  [5242] = {x=-104.947, y=80.94, z=66, rx=-180, rz=-143.366, shoulder=lefty, elbow=epositive, wrist=wpositive, fatherId=fReference[0]}
  [5243] = {x=-103.694, y=80.008, z=66, rx=-180, rz=-143.329, shoulder=lefty, elbow=epositive, wrist=wpositive, fatherId=fReference[0]}
  [5244] = {x=-102.442, y=79.076, z=66, rx=-180, rz=-143.293, shoulder=lefty, elbow=epositive, wrist=wpositive, fatherId=fReference[0]}
  [5245] = {x=-101.19, y=78.143, z=66, rx=-180, rz=-143.258, shoulder=lefty, elbow=epositive, wrist=wpositive, fatherId=fReference[0]}
  [5246] = {x=-99.938, y=77.208, z=66, rx=-180, rz=-143.223, shoulder=lefty, elbow=epositive, wrist=wpositive, fatherId=fReference[0]}
  [5247] = {x=-98.687, y=76.273, z=66, rx=-180, rz=-143.188, shoulder=lefty, elbow=epositive, wrist=wpositive, fatherId=fReference[0]}
  [5248] = {x=-97.437, y=75.337, z=66, rx=180, rz=-143.154, shoulder=lefty, elbow=epositive, wrist=wpositive, fatherId=fReference[0]}
  [5249] = {x=-96.186, y=74.4, z=66, rx=180, rz=-143.12, shoulder=lefty, elbow=epositive, wrist=wpositive, fatherId=fReference[0]}
  [5250] = {x=-94.936, y=73.462, z=66, rx=180, rz=-143.087, shoulder=lefty, elbow=epositive, wrist=wpositive, fatherId=fReference[0]}
  [5251] = {x=-93.686, y=72.523, z=66, rx=-180, rz=-143.054, shoulder=lefty, elbow=epositive, wrist=wpositive, fatherId=fReference[0]}
  [5252] = {x=-92.437, y=71.584, z=66, rx=180, rz=-143.022, shoulder=lefty, elbow=epositive, wrist=wpositive, fatherId=fReference[0]}
  [5253] = {x=-91.188, y=70.643, z=66, rx=-180, rz=-142.99, shoulder=lefty, elbow=epositive, wrist=wpositive, fatherId=fReference[0]}
  [5254] = {x=-89.939, y=69.702, z=66, rx=-180, rz=-142.959, shoulder=lefty, elbow=epositive, wrist=wpositive, fatherId=fReference[0]}
  [5255] = {x=-88.691, y=68.76, z=66, rx=-180, rz=-142.928, shoulder=lefty, elbow=epositive, wrist=wpositive, fatherId=fReference[0]}
  [5256] = {x=-87.443, y=67.817, z=66, rx=-180, rz=-142.897, shoulder=lefty, elbow=epositive, wrist=wpositive, fatherId=fReference[0]}
  [5257] = {x=-86.195, y=66.873, z=66, rx=180, rz=-142.867, shoulder=lefty, elbow=epositive, wrist=wpositive, fatherId=fReference[0]}
  [5258] = {x=-84.948, y=65.929, z=66, rx=-180, rz=-142.838, shoulder=lefty, elbow=epositive, wrist=wpositive, fatherId=fReference[0]}
  [5259] = {x=-83.701, y=64.984, z=66, rx=180, rz=-142.809, shoulder=lefty, elbow=epositive, wrist=wpositive, fatherId=fReference[0]}
  [5260] = {x=-82.454, y=64.038, z=66, rx=180, rz=-142.78, shoulder=lefty, elbow=epositive, wrist=wpositive, fatherId=fReference[0]}
  [5261] = {x=-81.208, y=63.091, z=66, rx=-180, rz=-142.752, shoulder=lefty, elbow=epositive, wrist=wpositive, fatherId=fReference[0]}
  [5262] = {x=-79.962, y=62.143, z=66, rx=-180, rz=-142.724, shoulder=lefty, elbow=epositive, wrist=wpositive, fatherId=fReference[0]}
  [5263] = {x=-78.716, y=61.195, z=66, rx=-180, rz=-142.697, shoulder=lefty, elbow=epositive, wrist=wpositive, fatherId=fReference[0]}
  [5264] = {x=-77.47, y=60.246, z=66, rx=-180, rz=-142.67, shoulder=lefty, elbow=epositive, wrist=wpositive, fatherId=fReference[0]}
  [5265] = {x=-76.225, y=59.297, z=66, rx=180, rz=-142.644, shoulder=lefty, elbow=epositive, wrist=wpositive, fatherId=fReference[0]}
  [5266] = {x=-74.98, y=58.346, z=66, rx=-180, rz=-142.618, shoulder=lefty, elbow=epositive, wrist=wpositive, fatherId=fReference[0]}
  [5267] = {x=-73.736, y=57.395, z=66, rx=180, rz=-142.592, shoulder=lefty, elbow=epositive, wrist=wpositive, fatherId=fReference[0]}
  [5268] = {x=-72.491, y=56.444, z=66, rx=-180, rz=-142.567, shoulder=lefty, elbow=epositive, wrist=wpositive, fatherId=fReference[0]}
  [5269] = {x=-71.247, y=55.491, z=66, rx=180, rz=-142.543, shoulder=lefty, elbow=epositive, wrist=wpositive, fatherId=fReference[0]}
  [5270] = {x=-70.003, y=54.538, z=66, rx=180, rz=-142.518, shoulder=lefty, elbow=epositive, wrist=wpositive, fatherId=fReference[0]}
  [5271] = {x=-68.76, y=53.585, z=66, rx=-180, rz=-142.495, shoulder=lefty, elbow=epositive, wrist=wpositive, fatherId=fReference[0]}
  [5272] = {x=-67.516, y=52.63, z=66, rx=-180, rz=-142.471, shoulder=lefty, elbow=epositive, wrist=wpositive, fatherId=fReference[0]}
  [5273] = {x=-66.273, y=51.676, z=66, rx=-180, rz=-142.449, shoulder=lefty, elbow=epositive, wrist=wpositive, fatherId=fReference[0]}
  [5274] = {x=-65.03, y=50.72, z=66, rx=-180, rz=-142.426, shoulder=lefty, elbow=epositive, wrist=wpositive, fatherId=fReference[0]}
  [5275] = {x=-63.788, y=49.764, z=66, rx=-180, rz=-142.404, shoulder=lefty, elbow=epositive, wrist=wpositive, fatherId=fReference[0]}
  [5276] = {x=-62.545, y=48.808, z=66, rx=-180, rz=-142.383, shoulder=lefty, elbow=epositive, wrist=wpositive, fatherId=fReference[0]}
  [5277] = {x=-61.303, y=47.85, z=66, rx=-180, rz=-142.362, shoulder=lefty, elbow=epositive, wrist=wpositive, fatherId=fReference[0]}
  [5278] = {x=-60.061, y=46.893, z=66, rx=-180, rz=-142.341, shoulder=lefty, elbow=epositive, wrist=wpositive, fatherId=fReference[0]}
  [5279] = {x=-58.82, y=45.934, z=66, rx=180, rz=-142.321, shoulder=lefty, elbow=epositive, wrist=wpositive, fatherId=fReference[0]}
  [5280] = {x=-57.578, y=44.976, z=66, rx=-180, rz=-142.301, shoulder=lefty, elbow=epositive, wrist=wpositive, fatherId=fReference[0]}
  [5281] = {x=-56.337, y=44.016, z=66, rx=180, rz=-142.282, shoulder=lefty, elbow=epositive, wrist=wpositive, fatherId=fReference[0]}
  [5282] = {x=-55.096, y=43.057, z=66, rx=-180, rz=-142.263, shoulder=lefty, elbow=epositive, wrist=wpositive, fatherId=fReference[0]}
  [5283] = {x=-53.855, y=42.096, z=66, rx=-180, rz=-142.244, shoulder=lefty, elbow=epositive, wrist=wpositive, fatherId=fReference[0]}
  [5284] = {x=-52.615, y=41.135, z=66, rx=-180, rz=-142.226, shoulder=lefty, elbow=epositive, wrist=wpositive, fatherId=fReference[0]}
  [5285] = {x=-51.374, y=40.174, z=66, rx=-180, rz=-142.209, shoulder=lefty, elbow=epositive, wrist=wpositive, fatherId=fReference[0]}
  [5286] = {x=-50.134, y=39.212, z=66, rx=-180, rz=-142.192, shoulder=lefty, elbow=epositive, wrist=wpositive, fatherId=fReference[0]}
  [5287] = {x=-48.894, y=38.25, z=66, rx=-180, rz=-142.175, shoulder=lefty, elbow=epositive, wrist=wpositive, fatherId=fReference[0]}
  [5288] = {x=-47.654, y=37.288, z=66, rx=-180, rz=-142.159, shoulder=lefty, elbow=epositive, wrist=wpositive, fatherId=fReference[0]}
  [5289] = {x=-46.414, y=36.325, z=66, rx=180, rz=-142.143, shoulder=lefty, elbow=epositive, wrist=wpositive, fatherId=fReference[0]}
  [5290] = {x=-45.175, y=35.361, z=66, rx=-180, rz=-142.127, shoulder=lefty, elbow=epositive, wrist=wpositive, fatherId=fReference[0]}
  [5291] = {x=-43.935, y=34.397, z=66, rx=180, rz=-142.112, shoulder=lefty, elbow=epositive, wrist=wpositive, fatherId=fReference[0]}
  [5292] = {x=-42.696, y=33.433, z=66, rx=180, rz=-142.098, shoulder=lefty, elbow=epositive, wrist=wpositive, fatherId=fReference[0]}
  [5293] = {x=-41.457, y=32.468, z=66, rx=180, rz=-142.083, shoulder=lefty, elbow=epositive, wrist=wpositive, fatherId=fReference[0]}
  [5294] = {x=-40.218, y=31.503, z=66, rx=-180, rz=-142.07, shoulder=lefty, elbow=epositive, wrist=wpositive, fatherId=fReference[0]}
  [5295] = {x=-38.979, y=30.538, z=66, rx=180, rz=-142.056, shoulder=lefty, elbow=epositive, wrist=wpositive, fatherId=fReference[0]}
  [5296] = {x=-37.74, y=29.572, z=66, rx=-180, rz=-142.044, shoulder=lefty, elbow=epositive, wrist=wpositive, fatherId=fReference[0]}
  [5297] = {x=-36.502, y=28.606, z=66, rx=-180, rz=-142.031, shoulder=lefty, elbow=epositive, wrist=wpositive, fatherId=fReference[0]}
  [5298] = {x=-35.263, y=27.639, z=66, rx=180, rz=-142.019, shoulder=lefty, elbow=epositive, wrist=wpositive, fatherId=fReference[0]}
  [5299] = {x=-34.025, y=26.672, z=66, rx=-180, rz=-142.007, shoulder=lefty, elbow=epositive, wrist=wpositive, fatherId=fReference[0]}
  [5300] = {x=-32.787, y=25.705, z=66, rx=-180, rz=-141.996, shoulder=lefty, elbow=epositive, wrist=wpositive, fatherId=fReference[0]}
  [5301] = {x=-31.549, y=24.738, z=66, rx=180, rz=-141.985, shoulder=lefty, elbow=epositive, wrist=wpositive, fatherId=fReference[0]}
  [5302] = {x=-30.311, y=23.77, z=66, rx=180, rz=-141.975, shoulder=lefty, elbow=epositive, wrist=wpositive, fatherId=fReference[0]}
  [5303] = {x=-29.073, y=22.802, z=66, rx=180, rz=-141.965, shoulder=lefty, elbow=epositive, wrist=wpositive, fatherId=fReference[0]}
  [5304] = {x=-27.835, y=21.834, z=66, rx=-180, rz=-141.956, shoulder=lefty, elbow=epositive, wrist=wpositive, fatherId=fReference[0]}
  [5305] = {x=-26.597, y=20.865, z=66, rx=-180, rz=-141.947, shoulder=lefty, elbow=epositive, wrist=wpositive, fatherId=fReference[0]}
  [5306] = {x=-25.36, y=19.896, z=66, rx=180, rz=-141.938, shoulder=lefty, elbow=epositive, wrist=wpositive, fatherId=fReference[0]}
  [5307] = {x=-24.122, y=18.927, z=66, rx=-180, rz=-141.93, shoulder=lefty, elbow=epositive, wrist=wpositive, fatherId=fReference[0]}
  [5308] = {x=-22.885, y=17.958, z=66, rx=180, rz=-141.922, shoulder=lefty, elbow=epositive, wrist=wpositive, fatherId=fReference[0]}
  [5309] = {x=-21.647, y=16.988, z=66, rx=-180, rz=-141.915, shoulder=lefty, elbow=epositive, wrist=wpositive, fatherId=fReference[0]}
  [5310] = {x=-20.41, y=16.019, z=66, rx=-180, rz=-141.908, shoulder=lefty, elbow=epositive, wrist=wpositive, fatherId=fReference[0]}
  [5311] = {x=-19.172, y=15.049, z=66, rx=-180, rz=-141.901, shoulder=lefty, elbow=epositive, wrist=wpositive, fatherId=fReference[0]}
  [5312] = {x=-17.935, y=14.079, z=66, rx=-180, rz=-141.895, shoulder=lefty, elbow=epositive, wrist=wpositive, fatherId=fReference[0]}
  [5313] = {x=-16.698, y=13.109, z=66, rx=180, rz=-141.889, shoulder=lefty, elbow=epositive, wrist=wpositive, fatherId=fReference[0]}
  [5314] = {x=-15.461, y=12.138, z=66, rx=-180, rz=-141.884, shoulder=lefty, elbow=epositive, wrist=wpositive, fatherId=fReference[0]}
  [5315] = {x=-14.224, y=11.168, z=66, rx=-180, rz=-141.879, shoulder=lefty, elbow=epositive, wrist=wpositive, fatherId=fReference[0]}
  [5316] = {x=-12.987, y=10.197, z=66, rx=-180, rz=-141.875, shoulder=lefty, elbow=epositive, wrist=wpositive, fatherId=fReference[0]}
  [5317] = {x=-11.75, y=9.226, z=66, rx=-180, rz=-141.871, shoulder=lefty, elbow=epositive, wrist=wpositive, fatherId=fReference[0]}
  [5318] = {x=-10.513, y=8.255, z=66, rx=-180, rz=-141.867, shoulder=lefty, elbow=epositive, wrist=wpositive, fatherId=fReference[0]}
  [5319] = {x=-9.276, y=7.284, z=66, rx=-180, rz=-141.864, shoulder=lefty, elbow=epositive, wrist=wpositive, fatherId=fReference[0]}
  [5320] = {x=-8.039, y=6.313, z=66, rx=180, rz=-141.862, shoulder=lefty, elbow=epositive, wrist=wpositive, fatherId=fReference[0]}
  [5321] = {x=-6.802, y=5.342, z=66, rx=-180, rz=-141.859, shoulder=lefty, elbow=epositive, wrist=wpositive, fatherId=fReference[0]}
  [5322] = {x=-5.565, y=4.37, z=66, rx=180, rz=-141.857, shoulder=lefty, elbow=epositive, wrist=wpositive, fatherId=fReference[0]}
  [5323] = {x=-4.328, y=3.399, z=66, rx=-180, rz=-141.856, shoulder=lefty, elbow=epositive, wrist=wpositive, fatherId=fReference[0]}
  [5324] = {x=-3.091, y=2.427, z=66, rx=-180, rz=-141.855, shoulder=lefty, elbow=epositive, wrist=wpositive, fatherId=fReference[0]}
  [5325] = {x=-1.854, y=1.456, z=66, rx=180, rz=-141.854, shoulder=lefty, elbow=epositive, wrist=wpositive, fatherId=fReference[0]}
  [5326] = {x=-0.617, y=0.484, z=66, rx=180, rz=-141.854, shoulder=lefty, elbow=epositive, wrist=wpositive, fatherId=fReference[0]}
  [5327] = {x=0.62, y=-0.487, z=66, rx=180, rz=-141.854, shoulder=lefty, elbow=epositive, wrist=wpositive, fatherId=fReference[0]}
  [5328] = {x=1.857, y=-1.459, z=66, rx=-180, rz=-141.855, shoulder=lefty, elbow=epositive, wrist=wpositive, fatherId=fReference[0]}
  [5329] = {x=3.094, y=-2.43, z=66, rx=180, rz=-141.856, shoulder=lefty, elbow=epositive, wrist=wpositive, fatherId=fReference[0]}
  [5330] = {x=4.331, y=-3.402, z=66, rx=-180, rz=-141.857, shoulder=lefty, elbow=epositive, wrist=wpositive, fatherId=fReference[0]}
  [5331] = {x=5.568, y=-4.373, z=66, rx=-180, rz=-141.859, shoulder=lefty, elbow=epositive, wrist=wpositive, fatherId=fReference[0]}
  [5332] = {x=6.805, y=-5.345, z=66, rx=180, rz=-141.862, shoulder=lefty, elbow=epositive, wrist=wpositive, fatherId=fReference[0]}
  [5333] = {x=8.043, y=-6.316, z=66, rx=180, rz=-141.864, shoulder=lefty, elbow=epositive, wrist=wpositive, fatherId=fReference[0]}
  [5334] = {x=9.28, y=-7.287, z=66, rx=180, rz=-141.867, shoulder=lefty, elbow=epositive, wrist=wpositive, fatherId=fReference[0]}
  [5335] = {x=10.517, y=-8.259, z=66, rx=180, rz=-141.871, shoulder=lefty, elbow=epositive, wrist=wpositive, fatherId=fReference[0]}
  [5336] = {x=11.754, y=-9.23, z=66, rx=-180, rz=-141.875, shoulder=lefty, elbow=epositive, wrist=wpositive, fatherId=fReference[0]}
  [5337] = {x=12.992, y=-10.201, z=66, rx=-180, rz=-141.879, shoulder=lefty, elbow=epositive, wrist=wpositive, fatherId=fReference[0]}
  [5338] = {x=14.229, y=-11.172, z=66, rx=180, rz=-141.884, shoulder=lefty, elbow=epositive, wrist=wpositive, fatherId=fReference[0]}
  [5339] = {x=15.467, y=-12.143, z=66, rx=-180, rz=-141.89, shoulder=lefty, elbow=epositive, wrist=wpositive, fatherId=fReference[0]}
  [5340] = {x=16.704, y=-13.113, z=66, rx=180, rz=-141.895, shoulder=lefty, elbow=epositive, wrist=wpositive, fatherId=fReference[0]}
  [5341] = {x=17.942, y=-14.084, z=66, rx=180, rz=-141.901, shoulder=lefty, elbow=epositive, wrist=wpositive, fatherId=fReference[0]}
  [5342] = {x=19.179, y=-15.054, z=66, rx=-180, rz=-141.908, shoulder=lefty, elbow=epositive, wrist=wpositive, fatherId=fReference[0]}
  [5343] = {x=20.417, y=-16.025, z=66, rx=-180, rz=-141.915, shoulder=lefty, elbow=epositive, wrist=wpositive, fatherId=fReference[0]}
  [5344] = {x=21.655, y=-16.995, z=66, rx=180, rz=-141.922, shoulder=lefty, elbow=epositive, wrist=wpositive, fatherId=fReference[0]}
  [5345] = {x=22.893, y=-17.965, z=66, rx=180, rz=-141.93, shoulder=lefty, elbow=epositive, wrist=wpositive, fatherId=fReference[0]}
  [5346] = {x=24.131, y=-18.934, z=66, rx=-180, rz=-141.938, shoulder=lefty, elbow=epositive, wrist=wpositive, fatherId=fReference[0]}
  [5347] = {x=25.369, y=-19.904, z=66, rx=-180, rz=-141.947, shoulder=lefty, elbow=epositive, wrist=wpositive, fatherId=fReference[0]}
  [5348] = {x=26.607, y=-20.873, z=66, rx=180, rz=-141.956, shoulder=lefty, elbow=epositive, wrist=wpositive, fatherId=fReference[0]}
  [5349] = {x=27.846, y=-21.842, z=66, rx=-180, rz=-141.965, shoulder=lefty, elbow=epositive, wrist=wpositive, fatherId=fReference[0]}
  [5350] = {x=29.084, y=-22.811, z=66, rx=-180, rz=-141.975, shoulder=lefty, elbow=epositive, wrist=wpositive, fatherId=fReference[0]}
  [5351] = {x=30.323, y=-23.779, z=66, rx=-180, rz=-141.986, shoulder=lefty, elbow=epositive, wrist=wpositive, fatherId=fReference[0]}
  [5352] = {x=31.561, y=-24.748, z=66, rx=-180, rz=-141.996, shoulder=lefty, elbow=epositive, wrist=wpositive, fatherId=fReference[0]}
  [5353] = {x=32.8, y=-25.716, z=66, rx=-180, rz=-142.008, shoulder=lefty, elbow=epositive, wrist=wpositive, fatherId=fReference[0]}
  [5354] = {x=34.039, y=-26.683, z=66, rx=180, rz=-142.019, shoulder=lefty, elbow=epositive, wrist=wpositive, fatherId=fReference[0]}
  [5355] = {x=35.278, y=-27.651, z=66, rx=-180, rz=-142.031, shoulder=lefty, elbow=epositive, wrist=wpositive, fatherId=fReference[0]}
  [5356] = {x=36.517, y=-28.618, z=66, rx=180, rz=-142.044, shoulder=lefty, elbow=epositive, wrist=wpositive, fatherId=fReference[0]}
  [5357] = {x=37.757, y=-29.585, z=66, rx=-180, rz=-142.057, shoulder=lefty, elbow=epositive, wrist=wpositive, fatherId=fReference[0]}
  [5358] = {x=38.996, y=-30.551, z=66, rx=-180, rz=-142.07, shoulder=lefty, elbow=epositive, wrist=wpositive, fatherId=fReference[0]}
  [5359] = {x=40.236, y=-31.517, z=66, rx=-180, rz=-142.084, shoulder=lefty, elbow=epositive, wrist=wpositive, fatherId=fReference[0]}
  [5360] = {x=41.476, y=-32.483, z=66, rx=-180, rz=-142.098, shoulder=lefty, elbow=epositive, wrist=wpositive, fatherId=fReference[0]}
  [5361] = {x=42.715, y=-33.448, z=66, rx=180, rz=-142.113, shoulder=lefty, elbow=epositive, wrist=wpositive, fatherId=fReference[0]}
  [5362] = {x=43.956, y=-34.413, z=66, rx=180, rz=-142.128, shoulder=lefty, elbow=epositive, wrist=wpositive, fatherId=fReference[0]}
  [5363] = {x=45.196, y=-35.377, z=66, rx=-180, rz=-142.143, shoulder=lefty, elbow=epositive, wrist=wpositive, fatherId=fReference[0]}
  [5364] = {x=46.436, y=-36.342, z=66, rx=-180, rz=-142.159, shoulder=lefty, elbow=epositive, wrist=wpositive, fatherId=fReference[0]}
  [5365] = {x=47.677, y=-37.305, z=66, rx=-180, rz=-142.175, shoulder=lefty, elbow=epositive, wrist=wpositive, fatherId=fReference[0]}
  [5366] = {x=48.917, y=-38.269, z=66, rx=180, rz=-142.192, shoulder=lefty, elbow=epositive, wrist=wpositive, fatherId=fReference[0]}
  [5367] = {x=50.158, y=-39.231, z=66, rx=180, rz=-142.209, shoulder=lefty, elbow=epositive, wrist=wpositive, fatherId=fReference[0]}
  [5368] = {x=51.399, y=-40.194, z=66, rx=180, rz=-142.227, shoulder=lefty, elbow=epositive, wrist=wpositive, fatherId=fReference[0]}
  [5369] = {x=52.641, y=-41.156, z=66, rx=-180, rz=-142.245, shoulder=lefty, elbow=epositive, wrist=wpositive, fatherId=fReference[0]}
  [5370] = {x=53.882, y=-42.117, z=66, rx=180, rz=-142.263, shoulder=lefty, elbow=epositive, wrist=wpositive, fatherId=fReference[0]}
  [5371] = {x=55.124, y=-43.078, z=66, rx=180, rz=-142.282, shoulder=lefty, elbow=epositive, wrist=wpositive, fatherId=fReference[0]}
  [5372] = {x=56.366, y=-44.038, z=66, rx=-180, rz=-142.302, shoulder=lefty, elbow=epositive, wrist=wpositive, fatherId=fReference[0]}
  [5373] = {x=57.608, y=-44.998, z=66, rx=180, rz=-142.321, shoulder=lefty, elbow=epositive, wrist=wpositive, fatherId=fReference[0]}
  [5374] = {x=58.85, y=-45.958, z=66, rx=-180, rz=-142.342, shoulder=lefty, elbow=epositive, wrist=wpositive, fatherId=fReference[0]}
  [5375] = {x=60.092, y=-46.916, z=66, rx=-180, rz=-142.362, shoulder=lefty, elbow=epositive, wrist=wpositive, fatherId=fReference[0]}
  [5376] = {x=61.335, y=-47.875, z=66, rx=180, rz=-142.383, shoulder=lefty, elbow=epositive, wrist=wpositive, fatherId=fReference[0]}
  [5377] = {x=62.578, y=-48.832, z=66, rx=-180, rz=-142.405, shoulder=lefty, elbow=epositive, wrist=wpositive, fatherId=fReference[0]}
  [5378] = {x=63.821, y=-49.79, z=66, rx=-180, rz=-142.427, shoulder=lefty, elbow=epositive, wrist=wpositive, fatherId=fReference[0]}
  [5379] = {x=65.064, y=-50.746, z=66, rx=180, rz=-142.449, shoulder=lefty, elbow=epositive, wrist=wpositive, fatherId=fReference[0]}
  [5380] = {x=66.308, y=-51.702, z=66, rx=-180, rz=-142.472, shoulder=lefty, elbow=epositive, wrist=wpositive, fatherId=fReference[0]}
  [5381] = {x=67.551, y=-52.657, z=66, rx=-180, rz=-142.496, shoulder=lefty, elbow=epositive, wrist=wpositive, fatherId=fReference[0]}
  [5382] = {x=68.795, y=-53.612, z=66, rx=-180, rz=-142.519, shoulder=lefty, elbow=epositive, wrist=wpositive, fatherId=fReference[0]}
  [5383] = {x=70.04, y=-54.566, z=66, rx=180, rz=-142.543, shoulder=lefty, elbow=epositive, wrist=wpositive, fatherId=fReference[0]}
  [5384] = {x=71.284, y=-55.519, z=66, rx=-180, rz=-142.568, shoulder=lefty, elbow=epositive, wrist=wpositive, fatherId=fReference[0]}
  [5385] = {x=72.529, y=-56.472, z=66, rx=-180, rz=-142.593, shoulder=lefty, elbow=epositive, wrist=wpositive, fatherId=fReference[0]}
  [5386] = {x=73.774, y=-57.424, z=66, rx=180, rz=-142.619, shoulder=lefty, elbow=epositive, wrist=wpositive, fatherId=fReference[0]}
  [5387] = {x=75.019, y=-58.376, z=66, rx=-180, rz=-142.645, shoulder=lefty, elbow=epositive, wrist=wpositive, fatherId=fReference[0]}
  [5388] = {x=76.264, y=-59.326, z=66, rx=-180, rz=-142.671, shoulder=lefty, elbow=epositive, wrist=wpositive, fatherId=fReference[0]}
  [5389] = {x=77.51, y=-60.276, z=66, rx=-180, rz=-142.698, shoulder=lefty, elbow=epositive, wrist=wpositive, fatherId=fReference[0]}
  [5390] = {x=78.756, y=-61.226, z=66, rx=-180, rz=-142.725, shoulder=lefty, elbow=epositive, wrist=wpositive, fatherId=fReference[0]}
  [5391] = {x=80.002, y=-62.174, z=66, rx=180, rz=-142.753, shoulder=lefty, elbow=epositive, wrist=wpositive, fatherId=fReference[0]}
  [5392] = {x=81.249, y=-63.122, z=66, rx=-180, rz=-142.781, shoulder=lefty, elbow=epositive, wrist=wpositive, fatherId=fReference[0]}
  [5393] = {x=82.496, y=-64.069, z=66, rx=180, rz=-142.81, shoulder=lefty, elbow=epositive, wrist=wpositive, fatherId=fReference[0]}
  [5394] = {x=83.743, y=-65.015, z=66, rx=180, rz=-142.839, shoulder=lefty, elbow=epositive, wrist=wpositive, fatherId=fReference[0]}
  [5395] = {x=84.99, y=-65.961, z=66, rx=-180, rz=-142.868, shoulder=lefty, elbow=epositive, wrist=wpositive, fatherId=fReference[0]}
  [5396] = {x=86.238, y=-66.905, z=66, rx=-180, rz=-142.898, shoulder=lefty, elbow=epositive, wrist=wpositive, fatherId=fReference[0]}
  [5397] = {x=87.486, y=-67.849, z=66, rx=-180, rz=-142.929, shoulder=lefty, elbow=epositive, wrist=wpositive, fatherId=fReference[0]}
  [5398] = {x=88.734, y=-68.792, z=66, rx=-180, rz=-142.96, shoulder=lefty, elbow=epositive, wrist=wpositive, fatherId=fReference[0]}
  [5399] = {x=89.982, y=-69.734, z=66, rx=-180, rz=-142.991, shoulder=lefty, elbow=epositive, wrist=wpositive, fatherId=fReference[0]}
  [5400] = {x=91.231, y=-70.676, z=66, rx=-180, rz=-143.023, shoulder=lefty, elbow=epositive, wrist=wpositive, fatherId=fReference[0]}
  [5401] = {x=92.48, y=-71.616, z=66, rx=180, rz=-143.055, shoulder=lefty, elbow=epositive, wrist=wpositive, fatherId=fReference[0]}
  [5402] = {x=93.73, y=-72.556, z=66, rx=-180, rz=-143.088, shoulder=lefty, elbow=epositive, wrist=wpositive, fatherId=fReference[0]}
  [5403] = {x=94.979, y=-73.495, z=66, rx=-180, rz=-143.121, shoulder=lefty, elbow=epositive, wrist=wpositive, fatherId=fReference[0]}
  [5404] = {x=96.23, y=-74.432, z=66, rx=-180, rz=-143.155, shoulder=lefty, elbow=epositive, wrist=wpositive, fatherId=fReference[0]}
  [5405] = {x=97.48, y=-75.369, z=66, rx=180, rz=-143.189, shoulder=lefty, elbow=epositive, wrist=wpositive, fatherId=fReference[0]}
  [5406] = {x=98.731, y=-76.305, z=66, rx=180, rz=-143.224, shoulder=lefty, elbow=epositive, wrist=wpositive, fatherId=fReference[0]}
  [5407] = {x=99.982, y=-77.24, z=66, rx=-180, rz=-143.259, shoulder=lefty, elbow=epositive, wrist=wpositive, fatherId=fReference[0]}
  [5408] = {x=101.233, y=-78.175, z=66, rx=180, rz=-143.294, shoulder=lefty, elbow=epositive, wrist=wpositive, fatherId=fReference[0]}
  [5409] = {x=102.485, y=-79.108, z=66, rx=-180, rz=-143.33, shoulder=lefty, elbow=epositive, wrist=wpositive, fatherId=fReference[0]}
  [5410] = {x=103.737, y=-80.04, z=66, rx=-180, rz=-143.367, shoulder=lefty, elbow=epositive, wrist=wpositive, fatherId=fReference[0]}
  [5411] = {x=104.989, y=-80.971, z=66, rx=180, rz=-143.404, shoulder=lefty, elbow=epositive, wrist=wpositive, fatherId=fReference[0]}
  [5412] = {x=106.242, y=-81.901, z=66, rx=180, rz=-143.441, shoulder=lefty, elbow=epositive, wrist=wpositive, fatherId=fReference[0]}
  [5413] = {x=107.495, y=-82.831, z=66, rx=180, rz=-143.479, shoulder=lefty, elbow=epositive, wrist=wpositive, fatherId=fReference[0]}
  [5414] = {x=108.748, y=-83.759, z=66, rx=-180, rz=-143.517, shoulder=lefty, elbow=epositive, wrist=wpositive, fatherId=fReference[0]}
  [5415] = {x=110.002, y=-84.686, z=66, rx=-180, rz=-143.556, shoulder=lefty, elbow=epositive, wrist=wpositive, fatherId=fReference[0]}
  [5416] = {x=111.256, y=-85.612, z=66, rx=-180, rz=-143.596, shoulder=lefty, elbow=epositive, wrist=wpositive, fatherId=fReference[0]}
  [5417] = {x=112.511, y=-86.537, z=66, rx=180, rz=-143.635, shoulder=lefty, elbow=epositive, wrist=wpositive, fatherId=fReference[0]}
  [5418] = {x=113.766, y=-87.461, z=66, rx=-180, rz=-143.676, shoulder=lefty, elbow=epositive, wrist=wpositive, fatherId=fReference[0]}
  [5419] = {x=115.021, y=-88.384, z=66, rx=-180, rz=-143.716, shoulder=lefty, elbow=epositive, wrist=wpositive, fatherId=fReference[0]}
  [5420] = {x=116.277, y=-89.306, z=66, rx=-180, rz=-143.758, shoulder=lefty, elbow=epositive, wrist=wpositive, fatherId=fReference[0]}
  [5421] = {x=117.533, y=-90.227, z=66, rx=180, rz=-143.799, shoulder=lefty, elbow=epositive, wrist=wpositive, fatherId=fReference[0]}
  [5422] = {x=118.789, y=-91.146, z=66, rx=180, rz=-143.842, shoulder=lefty, elbow=epositive, wrist=wpositive, fatherId=fReference[0]}
  [5423] = {x=120.046, y=-92.065, z=66, rx=180, rz=-143.884, shoulder=lefty, elbow=epositive, wrist=wpositive, fatherId=fReference[0]}
  [5424] = {x=121.304, y=-92.982, z=66, rx=180, rz=-143.927, shoulder=lefty, elbow=epositive, wrist=wpositive, fatherId=fReference[0]}
  [5425] = {x=122.561, y=-93.898, z=66, rx=180, rz=-143.971, shoulder=lefty, elbow=epositive, wrist=wpositive, fatherId=fReference[0]}
  [5426] = {x=123.819, y=-94.813, z=66, rx=-180, rz=-144.015, shoulder=lefty, elbow=epositive, wrist=wpositive, fatherId=fReference[0]}
  [5427] = {x=125.078, y=-95.727, z=66, rx=-180, rz=-144.06, shoulder=lefty, elbow=epositive, wrist=wpositive, fatherId=fReference[0]}
  [5428] = {x=126.337, y=-96.64, z=66, rx=180, rz=-144.105, shoulder=lefty, elbow=epositive, wrist=wpositive, fatherId=fReference[0]}
  [5429] = {x=127.596, y=-97.551, z=66, rx=-180, rz=-144.151, shoulder=lefty, elbow=epositive, wrist=wpositive, fatherId=fReference[0]}
  [5430] = {x=128.856, y=-98.461, z=66, rx=180, rz=-144.197, shoulder=lefty, elbow=epositive, wrist=wpositive, fatherId=fReference[0]}
  [5431] = {x=130.116, y=-99.37, z=66, rx=180, rz=-144.243, shoulder=lefty, elbow=epositive, wrist=wpositive, fatherId=fReference[0]}
  [5432] = {x=131.376, y=-100.278, z=66, rx=-180, rz=-144.291, shoulder=lefty, elbow=epositive, wrist=wpositive, fatherId=fReference[0]}
  [5433] = {x=132.637, y=-101.185, z=66, rx=-180, rz=-144.338, shoulder=lefty, elbow=epositive, wrist=wpositive, fatherId=fReference[0]}
  [5434] = {x=133.899, y=-102.09, z=66, rx=-180, rz=-144.386, shoulder=lefty, elbow=epositive, wrist=wpositive, fatherId=fReference[0]}
  [5435] = {x=135.161, y=-102.994, z=66, rx=-180, rz=-144.435, shoulder=lefty, elbow=epositive, wrist=wpositive, fatherId=fReference[0]}
  [5436] = {x=136.423, y=-103.896, z=66, rx=180, rz=-144.484, shoulder=lefty, elbow=epositive, wrist=wpositive, fatherId=fReference[0]}
  [5437] = {x=137.686, y=-104.798, z=66, rx=-180, rz=-144.534, shoulder=lefty, elbow=epositive, wrist=wpositive, fatherId=fReference[0]}
  [5438] = {x=138.949, y=-105.698, z=66, rx=180, rz=-144.584, shoulder=lefty, elbow=epositive, wrist=wpositive, fatherId=fReference[0]}
  [5439] = {x=140.213, y=-106.596, z=66, rx=180, rz=-144.634, shoulder=lefty, elbow=epositive, wrist=wpositive, fatherId=fReference[0]}
  [5440] = {x=141.477, y=-107.494, z=66, rx=180, rz=-144.686, shoulder=lefty, elbow=epositive, wrist=wpositive, fatherId=fReference[0]}
  [5441] = {x=142.742, y=-108.389, z=66, rx=-180, rz=-144.737, shoulder=lefty, elbow=epositive, wrist=wpositive, fatherId=fReference[0]}
  [5442] = {x=144.007, y=-109.284, z=66, rx=180, rz=-144.789, shoulder=lefty, elbow=epositive, wrist=wpositive, fatherId=fReference[0]}
  [5443] = {x=145.273, y=-110.177, z=66, rx=-180, rz=-144.842, shoulder=lefty, elbow=epositive, wrist=wpositive, fatherId=fReference[0]}
  [5444] = {x=146.539, y=-111.069, z=66, rx=-180, rz=-144.895, shoulder=lefty, elbow=epositive, wrist=wpositive, fatherId=fReference[0]}
  [5445] = {x=147.806, y=-111.959, z=66, rx=180, rz=-144.949, shoulder=lefty, elbow=epositive, wrist=wpositive, fatherId=fReference[0]}
  [5446] = {x=149.073, y=-112.848, z=66, rx=-180, rz=-145.003, shoulder=lefty, elbow=epositive, wrist=wpositive, fatherId=fReference[0]}
  [5447] = {x=150.34, y=-113.736, z=66, rx=180, rz=-145.058, shoulder=lefty, elbow=epositive, wrist=wpositive, fatherId=fReference[0]}
  [5448] = {x=151.608, y=-114.622, z=66, rx=180, rz=-145.113, shoulder=lefty, elbow=epositive, wrist=wpositive, fatherId=fReference[0]}
  [5449] = {x=152.877, y=-115.506, z=66, rx=-180, rz=-145.169, shoulder=lefty, elbow=epositive, wrist=wpositive, fatherId=fReference[0]}
  [5450] = {x=154.146, y=-116.389, z=66, rx=-180, rz=-145.225, shoulder=lefty, elbow=epositive, wrist=wpositive, fatherId=fReference[0]}
  [5451] = {x=155.416, y=-117.271, z=66, rx=180, rz=-145.282, shoulder=lefty, elbow=epositive, wrist=wpositive, fatherId=fReference[0]}
  [5452] = {x=156.686, y=-118.151, z=66, rx=180, rz=-145.34, shoulder=lefty, elbow=epositive, wrist=wpositive, fatherId=fReference[0]}
  [5453] = {x=157.957, y=-119.03, z=66, rx=-180, rz=-145.398, shoulder=lefty, elbow=epositive, wrist=wpositive, fatherId=fReference[0]}
  [5454] = {x=159.228, y=-119.907, z=66, rx=180, rz=-145.456, shoulder=lefty, elbow=epositive, wrist=wpositive, fatherId=fReference[0]}
  [5455] = {x=160.5, y=-120.782, z=66, rx=-180, rz=-145.515, shoulder=lefty, elbow=epositive, wrist=wpositive, fatherId=fReference[0]}
  [5456] = {x=161.772, y=-121.656, z=66, rx=-180, rz=-145.575, shoulder=lefty, elbow=epositive, wrist=wpositive, fatherId=fReference[0]}
  [5457] = {x=163.045, y=-122.529, z=66, rx=180, rz=-145.635, shoulder=lefty, elbow=epositive, wrist=wpositive, fatherId=fReference[0]}
  [5458] = {x=164.319, y=-123.4, z=66, rx=-180, rz=-145.695, shoulder=lefty, elbow=epositive, wrist=wpositive, fatherId=fReference[0]}
  [5459] = {x=165.593, y=-124.269, z=66, rx=-180, rz=-145.756, shoulder=lefty, elbow=epositive, wrist=wpositive, fatherId=fReference[0]}
  [5460] = {x=166.867, y=-125.136, z=66, rx=-180, rz=-145.818, shoulder=lefty, elbow=epositive, wrist=wpositive, fatherId=fReference[0]}
  [5461] = {x=168.142, y=-126.002, z=66, rx=180, rz=-145.88, shoulder=lefty, elbow=epositive, wrist=wpositive, fatherId=fReference[0]}
  [5462] = {x=169.418, y=-126.867, z=66, rx=-180, rz=-145.943, shoulder=lefty, elbow=epositive, wrist=wpositive, fatherId=fReference[0]}
  [5463] = {x=170.695, y=-127.73, z=66, rx=-180, rz=-146.006, shoulder=lefty, elbow=epositive, wrist=wpositive, fatherId=fReference[0]}
  [5464] = {x=171.971, y=-128.591, z=66, rx=180, rz=-146.07, shoulder=lefty, elbow=epositive, wrist=wpositive, fatherId=fReference[0]}
  [5465] = {x=173.249, y=-129.45, z=66, rx=-180, rz=-146.135, shoulder=lefty, elbow=epositive, wrist=wpositive, fatherId=fReference[0]}
  [5466] = {x=174.527, y=-130.308, z=66, rx=180, rz=-146.2, shoulder=lefty, elbow=epositive, wrist=wpositive, fatherId=fReference[0]}
  [5467] = {x=175.806, y=-131.164, z=66, rx=-180, rz=-146.265, shoulder=lefty, elbow=epositive, wrist=wpositive, fatherId=fReference[0]}
  [5468] = {x=177.085, y=-132.018, z=66, rx=-180, rz=-146.331, shoulder=lefty, elbow=epositive, wrist=wpositive, fatherId=fReference[0]}
  [5469] = {x=178.365, y=-132.871, z=66, rx=180, rz=-146.398, shoulder=lefty, elbow=epositive, wrist=wpositive, fatherId=fReference[0]}
  [5470] = {x=179.645, y=-133.721, z=66, rx=-180, rz=-146.465, shoulder=lefty, elbow=epositive, wrist=wpositive, fatherId=fReference[0]}
  [5471] = {x=180.927, y=-134.571, z=66, rx=180, rz=-146.533, shoulder=lefty, elbow=epositive, wrist=wpositive, fatherId=fReference[0]}
  [5472] = {x=182.208, y=-135.418, z=66, rx=180, rz=-146.601, shoulder=lefty, elbow=epositive, wrist=wpositive, fatherId=fReference[0]}
  [5473] = {x=183.491, y=-136.263, z=66, rx=-180, rz=-146.67, shoulder=lefty, elbow=epositive, wrist=wpositive, fatherId=fReference[0]}
  [5474] = {x=184.774, y=-137.107, z=66, rx=-180, rz=-146.74, shoulder=lefty, elbow=epositive, wrist=wpositive, fatherId=fReference[0]}
  [5475] = {x=186.057, y=-137.949, z=66, rx=-180, rz=-146.81, shoulder=lefty, elbow=epositive, wrist=wpositive, fatherId=fReference[0]}
  [5476] = {x=187.341, y=-138.789, z=66, rx=-180, rz=-146.881, shoulder=lefty, elbow=epositive, wrist=wpositive, fatherId=fReference[0]}
  [5477] = {x=188.626, y=-139.627, z=66, rx=180, rz=-146.952, shoulder=lefty, elbow=epositive, wrist=wpositive, fatherId=fReference[0]}
  [5478] = {x=189.912, y=-140.464, z=66, rx=-180, rz=-147.024, shoulder=lefty, elbow=epositive, wrist=wpositive, fatherId=fReference[0]}
  [5479] = {x=191.198, y=-141.298, z=66, rx=-180, rz=-147.096, shoulder=lefty, elbow=epositive, wrist=wpositive, fatherId=fReference[0]}
  [5480] = {x=192.485, y=-142.131, z=66, rx=-180, rz=-147.169, shoulder=lefty, elbow=epositive, wrist=wpositive, fatherId=fReference[0]}
  [5481] = {x=193.772, y=-142.961, z=66, rx=-180, rz=-147.243, shoulder=lefty, elbow=epositive, wrist=wpositive, fatherId=fReference[0]}
  [5482] = {x=195.06, y=-143.79, z=66, rx=-180, rz=-147.317, shoulder=lefty, elbow=epositive, wrist=wpositive, fatherId=fReference[0]}
  [5483] = {x=196.349, y=-144.617, z=66, rx=-180, rz=-147.392, shoulder=lefty, elbow=epositive, wrist=wpositive, fatherId=fReference[0]}
  [5484] = {x=197.639, y=-145.442, z=66, rx=-180, rz=-147.467, shoulder=lefty, elbow=epositive, wrist=wpositive, fatherId=fReference[0]}
  [5485] = {x=198.929, y=-146.265, z=66, rx=-180, rz=-147.543, shoulder=lefty, elbow=epositive, wrist=wpositive, fatherId=fReference[0]}
  [5486] = {x=200.219, y=-147.086, z=66, rx=-180, rz=-147.619, shoulder=lefty, elbow=epositive, wrist=wpositive, fatherId=fReference[0]}
  [5487] = {x=201.511, y=-147.905, z=66, rx=-180, rz=-147.697, shoulder=lefty, elbow=epositive, wrist=wpositive, fatherId=fReference[0]}
  [5488] = {x=202.803, y=-148.722, z=66, rx=-180, rz=-147.774, shoulder=lefty, elbow=epositive, wrist=wpositive, fatherId=fReference[0]}
  [5489] = {x=204.096, y=-149.536, z=66, rx=180, rz=-147.853, shoulder=lefty, elbow=epositive, wrist=wpositive, fatherId=fReference[0]}
  [5490] = {x=205.389, y=-150.349, z=66, rx=-180, rz=-147.931, shoulder=lefty, elbow=epositive, wrist=wpositive, fatherId=fReference[0]}
  [5491] = {x=206.683, y=-151.16, z=66, rx=-180, rz=-148.011, shoulder=lefty, elbow=epositive, wrist=wpositive, fatherId=fReference[0]}
  [5492] = {x=207.978, y=-151.969, z=66, rx=-180, rz=-148.091, shoulder=lefty, elbow=epositive, wrist=wpositive, fatherId=fReference[0]}
  [5493] = {x=209.273, y=-152.775, z=66, rx=-180, rz=-148.172, shoulder=lefty, elbow=epositive, wrist=wpositive, fatherId=fReference[0]}
  [5494] = {x=210.569, y=-153.58, z=66, rx=180, rz=-148.253, shoulder=lefty, elbow=epositive, wrist=wpositive, fatherId=fReference[0]}
  [5495] = {x=211.866, y=-154.382, z=66, rx=180, rz=-148.335, shoulder=lefty, elbow=epositive, wrist=wpositive, fatherId=fReference[0]}
  [5496] = {x=213.164, y=-155.183, z=66, rx=-180, rz=-148.418, shoulder=lefty, elbow=epositive, wrist=wpositive, fatherId=fReference[0]}
  [5497] = {x=214.462, y=-155.981, z=66, rx=180, rz=-148.501, shoulder=lefty, elbow=epositive, wrist=wpositive, fatherId=fReference[0]}
  [5498] = {x=215.761, y=-156.777, z=66, rx=180, rz=-148.585, shoulder=lefty, elbow=epositive, wrist=wpositive, fatherId=fReference[0]}
  [5499] = {x=217.06, y=-157.57, z=66, rx=-180, rz=-148.669, shoulder=lefty, elbow=epositive, wrist=wpositive, fatherId=fReference[0]}
  [5500] = {x=218.361, y=-158.362, z=66, rx=-180, rz=-148.754, shoulder=lefty, elbow=epositive, wrist=wpositive, fatherId=fReference[0]}
  [5501] = {x=219.662, y=-159.151, z=66, rx=-180, rz=-148.84, shoulder=lefty, elbow=epositive, wrist=wpositive, fatherId=fReference[0]}
  [5502] = {x=220.963, y=-159.938, z=66, rx=-180, rz=-148.926, shoulder=lefty, elbow=epositive, wrist=wpositive, fatherId=fReference[0]}
  [5503] = {x=222.266, y=-160.723, z=66, rx=-180, rz=-149.013, shoulder=lefty, elbow=epositive, wrist=wpositive, fatherId=fReference[0]}
  [5504] = {x=223.569, y=-161.506, z=66, rx=-180, rz=-149.101, shoulder=lefty, elbow=epositive, wrist=wpositive, fatherId=fReference[0]}
  [5505] = {x=224.872, y=-162.286, z=66, rx=-180, rz=-149.189, shoulder=lefty, elbow=epositive, wrist=wpositive, fatherId=fReference[0]}
  [5506] = {x=226.177, y=-163.064, z=66, rx=-180, rz=-149.278, shoulder=lefty, elbow=epositive, wrist=wpositive, fatherId=fReference[0]}
  [5507] = {x=227.482, y=-163.84, z=66, rx=-180, rz=-149.367, shoulder=lefty, elbow=epositive, wrist=wpositive, fatherId=fReference[0]}
  [5508] = {x=228.788, y=-164.613, z=66, rx=-180, rz=-149.458, shoulder=lefty, elbow=epositive, wrist=wpositive, fatherId=fReference[0]}
  [5509] = {x=230.095, y=-165.384, z=66, rx=-180, rz=-149.548, shoulder=lefty, elbow=epositive, wrist=wpositive, fatherId=fReference[0]}
  [5510] = {x=231.402, y=-166.152, z=66, rx=180, rz=-149.64, shoulder=lefty, elbow=epositive, wrist=wpositive, fatherId=fReference[0]}
  [5511] = {x=232.71, y=-166.919, z=66, rx=-180, rz=-149.732, shoulder=lefty, elbow=epositive, wrist=wpositive, fatherId=fReference[0]}
  [5512] = {x=234.019, y=-167.682, z=66, rx=-180, rz=-149.824, shoulder=lefty, elbow=epositive, wrist=wpositive, fatherId=fReference[0]}
  [5513] = {x=235.328, y=-168.444, z=66, rx=180, rz=-149.918, shoulder=lefty, elbow=epositive, wrist=wpositive, fatherId=fReference[0]}
  [5514] = {x=236.638, y=-169.203, z=66, rx=-180, rz=-150.012, shoulder=lefty, elbow=epositive, wrist=wpositive, fatherId=fReference[0]}
  [5515] = {x=237.949, y=-169.959, z=66, rx=180, rz=-150.106, shoulder=lefty, elbow=epositive, wrist=wpositive, fatherId=fReference[0]}
  [5516] = {x=239.261, y=-170.713, z=66, rx=180, rz=-150.202, shoulder=lefty, elbow=epositive, wrist=wpositive, fatherId=fReference[0]}
  [5517] = {x=240.573, y=-171.465, z=66, rx=-180, rz=-150.298, shoulder=lefty, elbow=epositive, wrist=wpositive, fatherId=fReference[0]}
  [5518] = {x=241.886, y=-172.214, z=66, rx=-180, rz=-150.394, shoulder=lefty, elbow=epositive, wrist=wpositive, fatherId=fReference[0]}
  [5519] = {x=243.2, y=-172.96, z=66, rx=180, rz=-150.491, shoulder=lefty, elbow=epositive, wrist=wpositive, fatherId=fReference[0]}
  [5520] = {x=244.514, y=-173.704, z=66, rx=-180, rz=-150.589, shoulder=lefty, elbow=epositive, wrist=wpositive, fatherId=fReference[0]}
  [5521] = {x=245.83, y=-174.446, z=66, rx=-180, rz=-150.688, shoulder=lefty, elbow=epositive, wrist=wpositive, fatherId=fReference[0]}
  [5522] = {x=247.146, y=-175.184, z=66, rx=-180, rz=-150.787, shoulder=lefty, elbow=epositive, wrist=wpositive, fatherId=fReference[0]}
  [5523] = {x=248.462, y=-175.921, z=66, rx=-180, rz=-150.887, shoulder=lefty, elbow=epositive, wrist=wpositive, fatherId=fReference[0]}
  [5524] = {x=249.78, y=-176.654, z=66, rx=180, rz=-150.988, shoulder=lefty, elbow=epositive, wrist=wpositive, fatherId=fReference[0]}
  [5525] = {x=251.098, y=-177.385, z=66, rx=-180, rz=-151.089, shoulder=lefty, elbow=epositive, wrist=wpositive, fatherId=fReference[0]}
  [5526] = {x=252.417, y=-178.114, z=66, rx=-180, rz=-151.191, shoulder=lefty, elbow=epositive, wrist=wpositive, fatherId=fReference[0]}
  [5527] = {x=253.736, y=-178.839, z=66, rx=180, rz=-151.293, shoulder=lefty, elbow=epositive, wrist=wpositive, fatherId=fReference[0]}
  [5528] = {x=255.056, y=-179.562, z=66, rx=-180, rz=-151.397, shoulder=lefty, elbow=epositive, wrist=wpositive, fatherId=fReference[0]}
  [5529] = {x=256.378, y=-180.283, z=66, rx=-180, rz=-151.501, shoulder=lefty, elbow=epositive, wrist=wpositive, fatherId=fReference[0]}
  [5530] = {x=257.699, y=-181, z=66, rx=-180, rz=-151.605, shoulder=lefty, elbow=epositive, wrist=wpositive, fatherId=fReference[0]}
  [5531] = {x=259.022, y=-181.715, z=66, rx=180, rz=-151.711, shoulder=lefty, elbow=epositive, wrist=wpositive, fatherId=fReference[0]}
  [5532] = {x=260.345, y=-182.427, z=66, rx=-180, rz=-151.817, shoulder=lefty, elbow=epositive, wrist=wpositive, fatherId=fReference[0]}
  [5533] = {x=261.669, y=-183.137, z=66, rx=180, rz=-151.923, shoulder=lefty, elbow=epositive, wrist=wpositive, fatherId=fReference[0]}
  [5534] = {x=262.994, y=-183.843, z=66, rx=180, rz=-152.031, shoulder=lefty, elbow=epositive, wrist=wpositive, fatherId=fReference[0]}
  [5535] = {x=264.319, y=-184.547, z=66, rx=180, rz=-152.139, shoulder=lefty, elbow=epositive, wrist=wpositive, fatherId=fReference[0]}
  [5536] = {x=265.645, y=-185.248, z=66, rx=-180, rz=-152.247, shoulder=lefty, elbow=epositive, wrist=wpositive, fatherId=fReference[0]}
  [5537] = {x=266.972, y=-185.946, z=66, rx=-180, rz=-152.357, shoulder=lefty, elbow=epositive, wrist=wpositive, fatherId=fReference[0]}
  [5538] = {x=268.3, y=-186.642, z=66, rx=-180, rz=-152.467, shoulder=lefty, elbow=epositive, wrist=wpositive, fatherId=fReference[0]}
  [5539] = {x=269.628, y=-187.334, z=66, rx=-180, rz=-152.578, shoulder=lefty, elbow=epositive, wrist=wpositive, fatherId=fReference[0]}
  [5540] = {x=270.957, y=-188.024, z=66, rx=-180, rz=-152.689, shoulder=lefty, elbow=epositive, wrist=wpositive, fatherId=fReference[0]}
  [5541] = {x=272.287, y=-188.711, z=66, rx=180, rz=-152.801, shoulder=lefty, elbow=epositive, wrist=wpositive, fatherId=fReference[0]}
  [5542] = {x=273.617, y=-189.394, z=66, rx=-180, rz=-152.914, shoulder=lefty, elbow=epositive, wrist=wpositive, fatherId=fReference[0]}
  [5543] = {x=274.948, y=-190.075, z=66, rx=-180, rz=-153.028, shoulder=lefty, elbow=epositive, wrist=wpositive, fatherId=fReference[0]}
  [5544] = {x=276.28, y=-190.753, z=66, rx=180, rz=-153.142, shoulder=lefty, elbow=epositive, wrist=wpositive, fatherId=fReference[0]}
  [5545] = {x=277.613, y=-191.428, z=66, rx=-180, rz=-153.257, shoulder=lefty, elbow=epositive, wrist=wpositive, fatherId=fReference[0]}
  [5546] = {x=278.947, y=-192.1, z=66, rx=-180, rz=-153.372, shoulder=lefty, elbow=epositive, wrist=wpositive, fatherId=fReference[0]}
  [5547] = {x=280.281, y=-192.769, z=66, rx=-180, rz=-153.489, shoulder=lefty, elbow=epositive, wrist=wpositive, fatherId=fReference[0]}
  [5548] = {x=281.616, y=-193.435, z=66, rx=180, rz=-153.606, shoulder=lefty, elbow=epositive, wrist=wpositive, fatherId=fReference[0]}
  [5549] = {x=282.951, y=-194.097, z=66, rx=-180, rz=-153.724, shoulder=lefty, elbow=epositive, wrist=wpositive, fatherId=fReference[0]}
  [5550] = {x=284.288, y=-194.757, z=66, rx=-180, rz=-153.842, shoulder=lefty, elbow=epositive, wrist=wpositive, fatherId=fReference[0]}
  [5551] = {x=285.625, y=-195.414, z=66, rx=-180, rz=-153.961, shoulder=lefty, elbow=epositive, wrist=wpositive, fatherId=fReference[0]}
  [5552] = {x=286.963, y=-196.068, z=66, rx=180, rz=-154.081, shoulder=lefty, elbow=epositive, wrist=wpositive, fatherId=fReference[0]}
  [5553] = {x=288.301, y=-196.718, z=66, rx=-180, rz=-154.202, shoulder=lefty, elbow=epositive, wrist=wpositive, fatherId=fReference[0]}
  [5554] = {x=289.64, y=-197.365, z=66, rx=-180, rz=-154.323, shoulder=lefty, elbow=epositive, wrist=wpositive, fatherId=fReference[0]}
  [5555] = {x=290.98, y=-198.01, z=66, rx=-180, rz=-154.445, shoulder=lefty, elbow=epositive, wrist=wpositive, fatherId=fReference[0]}
  [5556] = {x=292.321, y=-198.651, z=66, rx=-180, rz=-154.568, shoulder=lefty, elbow=epositive, wrist=wpositive, fatherId=fReference[0]}
  [5557] = {x=293.663, y=-199.289, z=66, rx=-180, rz=-154.691, shoulder=lefty, elbow=epositive, wrist=wpositive, fatherId=fReference[0]}
  [5558] = {x=295.005, y=-199.923, z=66, rx=180, rz=-154.815, shoulder=lefty, elbow=epositive, wrist=wpositive, fatherId=fReference[0]}
  [5559] = {x=296.348, y=-200.555, z=66, rx=180, rz=-154.94, shoulder=lefty, elbow=epositive, wrist=wpositive, fatherId=fReference[0]}
  [5560] = {x=297.691, y=-201.183, z=66, rx=-180, rz=-155.066, shoulder=lefty, elbow=epositive, wrist=wpositive, fatherId=fReference[0]}
  [5561] = {x=299.036, y=-201.808, z=66, rx=180, rz=-155.192, shoulder=lefty, elbow=epositive, wrist=wpositive, fatherId=fReference[0]}
  [5562] = {x=300.381, y=-202.43, z=66, rx=-180, rz=-155.319, shoulder=lefty, elbow=epositive, wrist=wpositive, fatherId=fReference[0]}
  [5563] = {x=301.727, y=-203.048, z=66, rx=180, rz=-155.447, shoulder=lefty, elbow=epositive, wrist=wpositive, fatherId=fReference[0]}
  [5564] = {x=303.073, y=-203.663, z=66, rx=180, rz=-155.575, shoulder=lefty, elbow=epositive, wrist=wpositive, fatherId=fReference[0]}
  [5565] = {x=304.421, y=-204.275, z=66, rx=-180, rz=-155.705, shoulder=lefty, elbow=epositive, wrist=wpositive, fatherId=fReference[0]}
  [5566] = {x=305.769, y=-204.884, z=66, rx=-180, rz=-155.835, shoulder=lefty, elbow=epositive, wrist=wpositive, fatherId=fReference[0]}
  [5567] = {x=307.117, y=-205.489, z=66, rx=180, rz=-155.965, shoulder=lefty, elbow=epositive, wrist=wpositive, fatherId=fReference[0]}
  [5568] = {x=308.467, y=-206.091, z=66, rx=-180, rz=-156.097, shoulder=lefty, elbow=epositive, wrist=wpositive, fatherId=fReference[0]}
  [5569] = {x=309.817, y=-206.689, z=66, rx=-180, rz=-156.229, shoulder=lefty, elbow=epositive, wrist=wpositive, fatherId=fReference[0]}
  [5570] = {x=311.168, y=-207.284, z=66, rx=180, rz=-156.361, shoulder=lefty, elbow=epositive, wrist=wpositive, fatherId=fReference[0]}
  [5571] = {x=312.519, y=-207.876, z=66, rx=-180, rz=-156.495, shoulder=lefty, elbow=epositive, wrist=wpositive, fatherId=fReference[0]}
  [5572] = {x=313.872, y=-208.464, z=66, rx=-180, rz=-156.629, shoulder=lefty, elbow=epositive, wrist=wpositive, fatherId=fReference[0]}
  [5573] = {x=315.225, y=-209.049, z=66, rx=-180, rz=-156.764, shoulder=lefty, elbow=epositive, wrist=wpositive, fatherId=fReference[0]}
  [5574] = {x=316.579, y=-209.63, z=66, rx=180, rz=-156.9, shoulder=lefty, elbow=epositive, wrist=wpositive, fatherId=fReference[0]}
  [5575] = {x=317.933, y=-210.208, z=66, rx=-180, rz=-157.036, shoulder=lefty, elbow=epositive, wrist=wpositive, fatherId=fReference[0]}
  [5576] = {x=319.288, y=-210.782, z=66, rx=-180, rz=-157.173, shoulder=lefty, elbow=epositive, wrist=wpositive, fatherId=fReference[0]}
  [5577] = {x=320.644, y=-211.353, z=66, rx=-180, rz=-157.311, shoulder=lefty, elbow=epositive, wrist=wpositive, fatherId=fReference[0]}
  [5578] = {x=322.001, y=-211.92, z=66, rx=-180, rz=-157.45, shoulder=lefty, elbow=epositive, wrist=wpositive, fatherId=fReference[0]}
  [5579] = {x=323.358, y=-212.483, z=66, rx=-180, rz=-157.589, shoulder=lefty, elbow=epositive, wrist=wpositive, fatherId=fReference[0]}
  [5580] = {x=324.716, y=-213.044, z=66, rx=-180, rz=-157.729, shoulder=lefty, elbow=epositive, wrist=wpositive, fatherId=fReference[0]}
  [5581] = {x=326.075, y=-213.6, z=66, rx=-180, rz=-157.87, shoulder=lefty, elbow=epositive, wrist=wpositive, fatherId=fReference[0]}
  [5582] = {x=327.435, y=-214.153, z=66, rx=-180, rz=-158.011, shoulder=lefty, elbow=epositive, wrist=wpositive, fatherId=fReference[0]}
  [5583] = {x=328.795, y=-214.702, z=66, rx=-180, rz=-158.153, shoulder=lefty, elbow=epositive, wrist=wpositive, fatherId=fReference[0]}
  [5584] = {x=330.156, y=-215.248, z=66, rx=-180, rz=-158.296, shoulder=lefty, elbow=epositive, wrist=wpositive, fatherId=fReference[0]}
  [5585] = {x=331.517, y=-215.79, z=66, rx=-180, rz=-158.44, shoulder=lefty, elbow=epositive, wrist=wpositive, fatherId=fReference[0]}
  [5586] = {x=332.88, y=-216.328, z=66, rx=-180, rz=-158.584, shoulder=lefty, elbow=epositive, wrist=wpositive, fatherId=fReference[0]}
  [5587] = {x=334.243, y=-216.863, z=66, rx=-180, rz=-158.729, shoulder=lefty, elbow=epositive, wrist=wpositive, fatherId=fReference[0]}
  [5588] = {x=335.607, y=-217.394, z=66, rx=-180, rz=-158.875, shoulder=lefty, elbow=epositive, wrist=wpositive, fatherId=fReference[0]}
  [5589] = {x=336.971, y=-217.921, z=66, rx=-180, rz=-159.022, shoulder=lefty, elbow=epositive, wrist=wpositive, fatherId=fReference[0]}
  [5590] = {x=338.336, y=-218.444, z=66, rx=-180, rz=-159.169, shoulder=lefty, elbow=epositive, wrist=wpositive, fatherId=fReference[0]}
  [5591] = {x=339.702, y=-218.964, z=66, rx=-180, rz=-159.317, shoulder=lefty, elbow=epositive, wrist=wpositive, fatherId=fReference[0]}
  [5592] = {x=341.069, y=-219.48, z=66, rx=180, rz=-159.465, shoulder=lefty, elbow=epositive, wrist=wpositive, fatherId=fReference[0]}
  [5593] = {x=342.436, y=-219.992, z=66, rx=-180, rz=-159.615, shoulder=lefty, elbow=epositive, wrist=wpositive, fatherId=fReference[0]}
  [5594] = {x=343.804, y=-220.5, z=66, rx=-180, rz=-159.765, shoulder=lefty, elbow=epositive, wrist=wpositive, fatherId=fReference[0]}
  [5595] = {x=345.173, y=-221.005, z=66, rx=-180, rz=-159.916, shoulder=lefty, elbow=epositive, wrist=wpositive, fatherId=fReference[0]}
  [5596] = {x=346.542, y=-221.506, z=66, rx=180, rz=-160.067, shoulder=lefty, elbow=epositive, wrist=wpositive, fatherId=fReference[0]}
  [5597] = {x=347.912, y=-222.002, z=66, rx=-180, rz=-160.219, shoulder=lefty, elbow=epositive, wrist=wpositive, fatherId=fReference[0]}
  [5598] = {x=349.283, y=-222.495, z=66, rx=180, rz=-160.372, shoulder=lefty, elbow=epositive, wrist=wpositive, fatherId=fReference[0]}
  [5599] = {x=350.655, y=-222.985, z=66, rx=-180, rz=-160.526, shoulder=lefty, elbow=epositive, wrist=wpositive, fatherId=fReference[0]}
  [5600] = {x=352.027, y=-223.47, z=66, rx=-180, rz=-160.68, shoulder=lefty, elbow=epositive, wrist=wpositive, fatherId=fReference[0]}
  [5601] = {x=353.4, y=-223.951, z=66, rx=-180, rz=-160.835, shoulder=lefty, elbow=epositive, wrist=wpositive, fatherId=fReference[0]}
  [5602] = {x=354.773, y=-224.429, z=66, rx=180, rz=-160.991, shoulder=lefty, elbow=epositive, wrist=wpositive, fatherId=fReference[0]}
  [5603] = {x=356.148, y=-224.902, z=66, rx=180, rz=-161.147, shoulder=lefty, elbow=epositive, wrist=wpositive, fatherId=fReference[0]}
  [5604] = {x=357.523, y=-225.371, z=66, rx=-180, rz=-161.304, shoulder=lefty, elbow=epositive, wrist=wpositive, fatherId=fReference[0]}
  [5605] = {x=358.898, y=-225.837, z=66, rx=-180, rz=-161.462, shoulder=lefty, elbow=epositive, wrist=wpositive, fatherId=fReference[0]}
  [5606] = {x=360.275, y=-226.298, z=66, rx=-180, rz=-161.621, shoulder=lefty, elbow=epositive, wrist=wpositive, fatherId=fReference[0]}
  [5607] = {x=361.652, y=-226.756, z=66, rx=180, rz=-161.78, shoulder=lefty, elbow=epositive, wrist=wpositive, fatherId=fReference[0]}
  [5608] = {x=363.029, y=-227.209, z=66, rx=-180, rz=-161.94, shoulder=lefty, elbow=epositive, wrist=wpositive, fatherId=fReference[0]}
  [5609] = {x=364.407, y=-227.659, z=66, rx=180, rz=-162.1, shoulder=lefty, elbow=epositive, wrist=wpositive, fatherId=fReference[0]}
  [5610] = {x=365.786, y=-228.104, z=66, rx=-180, rz=-162.262, shoulder=lefty, elbow=epositive, wrist=wpositive, fatherId=fReference[0]}
  [5611] = {x=367.166, y=-228.546, z=66, rx=-180, rz=-162.424, shoulder=lefty, elbow=epositive, wrist=wpositive, fatherId=fReference[0]}
  [5612] = {x=368.546, y=-228.983, z=66, rx=-180, rz=-162.586, shoulder=lefty, elbow=epositive, wrist=wpositive, fatherId=fReference[0]}
  [5613] = {x=369.927, y=-229.416, z=66, rx=180, rz=-162.75, shoulder=lefty, elbow=epositive, wrist=wpositive, fatherId=fReference[0]}
  [5614] = {x=371.309, y=-229.845, z=66, rx=180, rz=-162.913, shoulder=lefty, elbow=epositive, wrist=wpositive, fatherId=fReference[0]}
  [5615] = {x=372.691, y=-230.27, z=66, rx=-180, rz=-163.078, shoulder=lefty, elbow=epositive, wrist=wpositive, fatherId=fReference[0]}
  [5616] = {x=374.074, y=-230.69, z=66, rx=-180, rz=-163.243, shoulder=lefty, elbow=epositive, wrist=wpositive, fatherId=fReference[0]}
  [5617] = {x=375.457, y=-231.107, z=66, rx=-180, rz=-163.409, shoulder=lefty, elbow=epositive, wrist=wpositive, fatherId=fReference[0]}
  [5618] = {x=376.841, y=-231.519, z=66, rx=-180, rz=-163.576, shoulder=lefty, elbow=epositive, wrist=wpositive, fatherId=fReference[0]}
  [5619] = {x=378.226, y=-231.928, z=66, rx=-180, rz=-163.743, shoulder=lefty, elbow=epositive, wrist=wpositive, fatherId=fReference[0]}
  [5620] = {x=379.611, y=-232.331, z=66, rx=-180, rz=-163.911, shoulder=lefty, elbow=epositive, wrist=wpositive, fatherId=fReference[0]}
  [5621] = {x=380.997, y=-232.731, z=66, rx=-180, rz=-164.08, shoulder=lefty, elbow=epositive, wrist=wpositive, fatherId=fReference[0]}
  [5622] = {x=382.384, y=-233.127, z=66, rx=180, rz=-164.249, shoulder=lefty, elbow=epositive, wrist=wpositive, fatherId=fReference[0]}
  [5623] = {x=383.771, y=-233.518, z=66, rx=180, rz=-164.419, shoulder=lefty, elbow=epositive, wrist=wpositive, fatherId=fReference[0]}
  [5624] = {x=385.159, y=-233.905, z=66, rx=180, rz=-164.589, shoulder=lefty, elbow=epositive, wrist=wpositive, fatherId=fReference[0]}
  [5625] = {x=386.547, y=-234.288, z=66, rx=180, rz=-164.76, shoulder=lefty, elbow=epositive, wrist=wpositive, fatherId=fReference[0]}
  [5626] = {x=387.936, y=-234.666, z=66, rx=180, rz=-164.932, shoulder=lefty, elbow=epositive, wrist=wpositive, fatherId=fReference[0]}
  [5627] = {x=389.325, y=-235.04, z=66, rx=180, rz=-165.105, shoulder=lefty, elbow=epositive, wrist=wpositive, fatherId=fReference[0]}
  [5628] = {x=390.715, y=-235.41, z=66, rx=-180, rz=-165.277, shoulder=lefty, elbow=epositive, wrist=wpositive, fatherId=fReference[0]}
  [5629] = {x=392.106, y=-235.775, z=66, rx=-180, rz=-165.451, shoulder=lefty, elbow=epositive, wrist=wpositive, fatherId=fReference[0]}
  [5630] = {x=393.497, y=-236.136, z=66, rx=180, rz=-165.625, shoulder=lefty, elbow=epositive, wrist=wpositive, fatherId=fReference[0]}
  [5631] = {x=394.889, y=-236.493, z=66, rx=-180, rz=-165.8, shoulder=lefty, elbow=epositive, wrist=wpositive, fatherId=fReference[0]}
  [5632] = {x=396.281, y=-236.845, z=66, rx=180, rz=-165.976, shoulder=lefty, elbow=epositive, wrist=wpositive, fatherId=fReference[0]}
  [5633] = {x=397.674, y=-237.193, z=66, rx=-180, rz=-166.152, shoulder=lefty, elbow=epositive, wrist=wpositive, fatherId=fReference[0]}
  [5634] = {x=399.068, y=-237.537, z=66, rx=180, rz=-166.328, shoulder=lefty, elbow=epositive, wrist=wpositive, fatherId=fReference[0]}
  [5635] = {x=400.462, y=-237.876, z=66, rx=180, rz=-166.505, shoulder=lefty, elbow=epositive, wrist=wpositive, fatherId=fReference[0]}
  [5636] = {x=401.856, y=-238.21, z=66, rx=-180, rz=-166.683, shoulder=lefty, elbow=epositive, wrist=wpositive, fatherId=fReference[0]}
  [5637] = {x=403.251, y=-238.541, z=66, rx=-180, rz=-166.861, shoulder=lefty, elbow=epositive, wrist=wpositive, fatherId=fReference[0]}
  [5638] = {x=404.647, y=-238.866, z=66, rx=-180, rz=-167.04, shoulder=lefty, elbow=epositive, wrist=wpositive, fatherId=fReference[0]}
  [5639] = {x=406.043, y=-239.188, z=66, rx=180, rz=-167.22, shoulder=lefty, elbow=epositive, wrist=wpositive, fatherId=fReference[0]}
  [5640] = {x=407.439, y=-239.505, z=66, rx=-180, rz=-167.4, shoulder=lefty, elbow=epositive, wrist=wpositive, fatherId=fReference[0]}
  [5641] = {x=408.836, y=-239.817, z=66, rx=180, rz=-167.581, shoulder=lefty, elbow=epositive, wrist=wpositive, fatherId=fReference[0]}
  [5642] = {x=410.234, y=-240.125, z=66, rx=-180, rz=-167.762, shoulder=lefty, elbow=epositive, wrist=wpositive, fatherId=fReference[0]}
  [5643] = {x=411.632, y=-240.428, z=66, rx=-180, rz=-167.943, shoulder=lefty, elbow=epositive, wrist=wpositive, fatherId=fReference[0]}
  [5644] = {x=413.031, y=-240.727, z=66, rx=180, rz=-168.126, shoulder=lefty, elbow=epositive, wrist=wpositive, fatherId=fReference[0]}
  [5645] = {x=414.43, y=-241.021, z=66, rx=-180, rz=-168.308, shoulder=lefty, elbow=epositive, wrist=wpositive, fatherId=fReference[0]}
  [5646] = {x=415.829, y=-241.31, z=66, rx=-180, rz=-168.492, shoulder=lefty, elbow=epositive, wrist=wpositive, fatherId=fReference[0]}
  [5647] = {x=417.229, y=-241.595, z=66, rx=-180, rz=-168.675, shoulder=lefty, elbow=epositive, wrist=wpositive, fatherId=fReference[0]}
  [5648] = {x=418.63, y=-241.876, z=66, rx=180, rz=-168.86, shoulder=lefty, elbow=epositive, wrist=wpositive, fatherId=fReference[0]}
  [5649] = {x=420.031, y=-242.152, z=66, rx=180, rz=-169.045, shoulder=lefty, elbow=epositive, wrist=wpositive, fatherId=fReference[0]}
  [5650] = {x=421.432, y=-242.423, z=66, rx=180, rz=-169.23, shoulder=lefty, elbow=epositive, wrist=wpositive, fatherId=fReference[0]}
  [5651] = {x=422.834, y=-242.69, z=66, rx=180, rz=-169.416, shoulder=lefty, elbow=epositive, wrist=wpositive, fatherId=fReference[0]}
  [5652] = {x=424.236, y=-242.952, z=66, rx=180, rz=-169.602, shoulder=lefty, elbow=epositive, wrist=wpositive, fatherId=fReference[0]}
  [5653] = {x=425.639, y=-243.209, z=66, rx=-180, rz=-169.789, shoulder=lefty, elbow=epositive, wrist=wpositive, fatherId=fReference[0]}
  [5654] = {x=427.042, y=-243.462, z=66, rx=180, rz=-169.976, shoulder=lefty, elbow=epositive, wrist=wpositive, fatherId=fReference[0]}
  [5655] = {x=428.445, y=-243.71, z=66, rx=-180, rz=-170.164, shoulder=lefty, elbow=epositive, wrist=wpositive, fatherId=fReference[0]}
  [5656] = {x=429.849, y=-243.953, z=66, rx=-180, rz=-170.352, shoulder=lefty, elbow=epositive, wrist=wpositive, fatherId=fReference[0]}
  [5657] = {x=431.254, y=-244.192, z=66, rx=180, rz=-170.54, shoulder=lefty, elbow=epositive, wrist=wpositive, fatherId=fReference[0]}
  [5658] = {x=432.658, y=-244.426, z=66, rx=-180, rz=-170.729, shoulder=lefty, elbow=epositive, wrist=wpositive, fatherId=fReference[0]}
  [5659] = {x=434.064, y=-244.655, z=66, rx=180, rz=-170.919, shoulder=lefty, elbow=epositive, wrist=wpositive, fatherId=fReference[0]}
  [5660] = {x=435.469, y=-244.88, z=66, rx=180, rz=-171.109, shoulder=lefty, elbow=epositive, wrist=wpositive, fatherId=fReference[0]}
  [5661] = {x=436.875, y=-245.1, z=66, rx=180, rz=-171.299, shoulder=lefty, elbow=epositive, wrist=wpositive, fatherId=fReference[0]}
  [5662] = {x=438.281, y=-245.315, z=66, rx=180, rz=-171.49, shoulder=lefty, elbow=epositive, wrist=wpositive, fatherId=fReference[0]}
  [5663] = {x=439.688, y=-245.526, z=66, rx=180, rz=-171.681, shoulder=lefty, elbow=epositive, wrist=wpositive, fatherId=fReference[0]}
  [5664] = {x=441.095, y=-245.731, z=66, rx=180, rz=-171.873, shoulder=lefty, elbow=epositive, wrist=wpositive, fatherId=fReference[0]}
  [5665] = {x=442.502, y=-245.932, z=66, rx=-180, rz=-172.065, shoulder=lefty, elbow=epositive, wrist=wpositive, fatherId=fReference[0]}
  [5666] = {x=443.91, y=-246.129, z=66, rx=-180, rz=-172.257, shoulder=lefty, elbow=epositive, wrist=wpositive, fatherId=fReference[0]}
  [5667] = {x=445.318, y=-246.32, z=66, rx=180, rz=-172.449, shoulder=lefty, elbow=epositive, wrist=wpositive, fatherId=fReference[0]}
  [5668] = {x=446.726, y=-246.507, z=66, rx=180, rz=-172.643, shoulder=lefty, elbow=epositive, wrist=wpositive, fatherId=fReference[0]}
  [5669] = {x=448.134, y=-246.689, z=66, rx=-180, rz=-172.836, shoulder=lefty, elbow=epositive, wrist=wpositive, fatherId=fReference[0]}
  [5670] = {x=449.543, y=-246.866, z=66, rx=180, rz=-173.03, shoulder=lefty, elbow=epositive, wrist=wpositive, fatherId=fReference[0]}
  [5671] = {x=450.953, y=-247.038, z=66, rx=-180, rz=-173.224, shoulder=lefty, elbow=epositive, wrist=wpositive, fatherId=fReference[0]}
  [5672] = {x=452.362, y=-247.205, z=66, rx=-180, rz=-173.418, shoulder=lefty, elbow=epositive, wrist=wpositive, fatherId=fReference[0]}
  [5673] = {x=453.772, y=-247.368, z=66, rx=180, rz=-173.613, shoulder=lefty, elbow=epositive, wrist=wpositive, fatherId=fReference[0]}
  [5674] = {x=455.182, y=-247.526, z=66, rx=180, rz=-173.808, shoulder=lefty, elbow=epositive, wrist=wpositive, fatherId=fReference[0]}
  [5675] = {x=456.592, y=-247.679, z=66, rx=-180, rz=-174.003, shoulder=lefty, elbow=epositive, wrist=wpositive, fatherId=fReference[0]}
  [5676] = {x=458.003, y=-247.827, z=66, rx=-180, rz=-174.199, shoulder=lefty, elbow=epositive, wrist=wpositive, fatherId=fReference[0]}
  [5677] = {x=459.414, y=-247.971, z=66, rx=-180, rz=-174.395, shoulder=lefty, elbow=epositive, wrist=wpositive, fatherId=fReference[0]}
  [5678] = {x=460.825, y=-248.109, z=66, rx=-180, rz=-174.591, shoulder=lefty, elbow=epositive, wrist=wpositive, fatherId=fReference[0]}
  [5679] = {x=462.236, y=-248.243, z=66, rx=180, rz=-174.787, shoulder=lefty, elbow=epositive, wrist=wpositive, fatherId=fReference[0]}
  [5680] = {x=463.647, y=-248.371, z=66, rx=-180, rz=-174.984, shoulder=lefty, elbow=epositive, wrist=wpositive, fatherId=fReference[0]}
  [5681] = {x=465.059, y=-248.495, z=66, rx=180, rz=-175.181, shoulder=lefty, elbow=epositive, wrist=wpositive, fatherId=fReference[0]}
  [5682] = {x=466.471, y=-248.614, z=66, rx=-180, rz=-175.378, shoulder=lefty, elbow=epositive, wrist=wpositive, fatherId=fReference[0]}
  [5683] = {x=467.883, y=-248.729, z=66, rx=180, rz=-175.575, shoulder=lefty, elbow=epositive, wrist=wpositive, fatherId=fReference[0]}
  [5684] = {x=469.296, y=-248.838, z=66, rx=-180, rz=-175.773, shoulder=lefty, elbow=epositive, wrist=wpositive, fatherId=fReference[0]}
  [5685] = {x=470.708, y=-248.942, z=66, rx=-180, rz=-175.971, shoulder=lefty, elbow=epositive, wrist=wpositive, fatherId=fReference[0]}
  [5686] = {x=472.121, y=-249.042, z=66, rx=-180, rz=-176.169, shoulder=lefty, elbow=epositive, wrist=wpositive, fatherId=fReference[0]}
  [5687] = {x=473.534, y=-249.136, z=66, rx=-180, rz=-176.367, shoulder=lefty, elbow=epositive, wrist=wpositive, fatherId=fReference[0]}
  [5688] = {x=474.947, y=-249.226, z=66, rx=-180, rz=-176.566, shoulder=lefty, elbow=epositive, wrist=wpositive, fatherId=fReference[0]}
  [5689] = {x=476.36, y=-249.311, z=66, rx=180, rz=-176.764, shoulder=lefty, elbow=epositive, wrist=wpositive, fatherId=fReference[0]}
  [5690] = {x=477.773, y=-249.391, z=66, rx=180, rz=-176.963, shoulder=lefty, elbow=epositive, wrist=wpositive, fatherId=fReference[0]}
  [5691] = {x=479.187, y=-249.466, z=66, rx=-180, rz=-177.162, shoulder=lefty, elbow=epositive, wrist=wpositive, fatherId=fReference[0]}
  [5692] = {x=480.6, y=-249.536, z=66, rx=-180, rz=-177.361, shoulder=lefty, elbow=epositive, wrist=wpositive, fatherId=fReference[0]}
  [5693] = {x=482.014, y=-249.601, z=66, rx=180, rz=-177.56, shoulder=lefty, elbow=epositive, wrist=wpositive, fatherId=fReference[0]}
  [5694] = {x=483.428, y=-249.661, z=66, rx=180, rz=-177.759, shoulder=lefty, elbow=epositive, wrist=wpositive, fatherId=fReference[0]}
  [5695] = {x=484.841, y=-249.717, z=66, rx=180, rz=-177.959, shoulder=lefty, elbow=epositive, wrist=wpositive, fatherId=fReference[0]}
  [5696] = {x=486.255, y=-249.767, z=66, rx=-180, rz=-178.158, shoulder=lefty, elbow=epositive, wrist=wpositive, fatherId=fReference[0]}
  [5697] = {x=487.669, y=-249.812, z=66, rx=180, rz=-178.358, shoulder=lefty, elbow=epositive, wrist=wpositive, fatherId=fReference[0]}
  [5698] = {x=489.084, y=-249.853, z=66, rx=180, rz=-178.557, shoulder=lefty, elbow=epositive, wrist=wpositive, fatherId=fReference[0]}
  [5699] = {x=490.498, y=-249.889, z=66, rx=180, rz=-178.757, shoulder=lefty, elbow=epositive, wrist=wpositive, fatherId=fReference[0]}
  [5700] = {x=491.912, y=-249.919, z=66, rx=180, rz=-178.957, shoulder=lefty, elbow=epositive, wrist=wpositive, fatherId=fReference[0]}
  [5701] = {x=493.326, y=-249.945, z=66, rx=180, rz=-179.157, shoulder=lefty, elbow=epositive, wrist=wpositive, fatherId=fReference[0]}
  [5702] = {x=494.741, y=-249.966, z=66, rx=180, rz=-179.357, shoulder=lefty, elbow=epositive, wrist=wpositive, fatherId=fReference[0]}
  [5703] = {x=496.155, y=-249.982, z=66, rx=-180, rz=-179.557, shoulder=lefty, elbow=epositive, wrist=wpositive, fatherId=fReference[0]}
  [5704] = {x=497.569, y=-249.993, z=66, rx=180, rz=-179.756, shoulder=lefty, elbow=epositive, wrist=wpositive, fatherId=fReference[0]}
  [5705] = {x=498.984, y=-249.999, z=66, rx=180, rz=-179.956, shoulder=lefty, elbow=epositive, wrist=wpositive, fatherId=fReference[0]}
  [5706] = {x=500.398, y=-250, z=66, rx=180, rz=179.844, shoulder=lefty, elbow=epositive, wrist=wpositive, fatherId=fReference[0]}
  [5707] = {x=501.812, y=-249.996, z=66, rx=180, rz=179.644, shoulder=lefty, elbow=epositive, wrist=wpositive, fatherId=fReference[0]}
  [5708] = {x=503.227, y=-249.987, z=66, rx=180, rz=179.444, shoulder=lefty, elbow=epositive, wrist=wpositive, fatherId=fReference[0]}
  [5709] = {x=504.641, y=-249.973, z=66, rx=-180, rz=179.244, shoulder=lefty, elbow=epositive, wrist=wpositive, fatherId=fReference[0]}
  [5710] = {x=506.055, y=-249.955, z=66, rx=-180, rz=179.044, shoulder=lefty, elbow=epositive, wrist=wpositive, fatherId=fReference[0]}
  [5711] = {x=507.47, y=-249.931, z=66, rx=180, rz=178.844, shoulder=lefty, elbow=epositive, wrist=wpositive, fatherId=fReference[0]}
  [5712] = {x=508.884, y=-249.903, z=66, rx=-180, rz=178.645, shoulder=lefty, elbow=epositive, wrist=wpositive, fatherId=fReference[0]}
  [5713] = {x=510.298, y=-249.869, z=66, rx=-180, rz=178.445, shoulder=lefty, elbow=epositive, wrist=wpositive, fatherId=fReference[0]}
  [5714] = {x=511.712, y=-249.831, z=66, rx=-180, rz=178.245, shoulder=lefty, elbow=epositive, wrist=wpositive, fatherId=fReference[0]}
  [5715] = {x=513.126, y=-249.787, z=66, rx=-180, rz=178.046, shoulder=lefty, elbow=epositive, wrist=wpositive, fatherId=fReference[0]}
  [5716] = {x=514.54, y=-249.739, z=66, rx=180, rz=177.846, shoulder=lefty, elbow=epositive, wrist=wpositive, fatherId=fReference[0]}
  [5717] = {x=515.954, y=-249.686, z=66, rx=-180, rz=177.647, shoulder=lefty, elbow=epositive, wrist=wpositive, fatherId=fReference[0]}
  [5718] = {x=517.368, y=-249.628, z=66, rx=-180, rz=177.448, shoulder=lefty, elbow=epositive, wrist=wpositive, fatherId=fReference[0]}
  [5719] = {x=518.782, y=-249.565, z=66, rx=-180, rz=177.249, shoulder=lefty, elbow=epositive, wrist=wpositive, fatherId=fReference[0]}
  [5720] = {x=520.195, y=-249.497, z=66, rx=-180, rz=177.05, shoulder=lefty, elbow=epositive, wrist=wpositive, fatherId=fReference[0]}
  [5721] = {x=521.609, y=-249.424, z=66, rx=180, rz=176.851, shoulder=lefty, elbow=epositive, wrist=wpositive, fatherId=fReference[0]}
  [5722] = {x=523.022, y=-249.346, z=66, rx=180, rz=176.652, shoulder=lefty, elbow=epositive, wrist=wpositive, fatherId=fReference[0]}
  [5723] = {x=524.435, y=-249.264, z=66, rx=-180, rz=176.454, shoulder=lefty, elbow=epositive, wrist=wpositive, fatherId=fReference[0]}
  [5724] = {x=525.848, y=-249.176, z=66, rx=-180, rz=176.256, shoulder=lefty, elbow=epositive, wrist=wpositive, fatherId=fReference[0]}
  [5725] = {x=527.261, y=-249.084, z=66, rx=-180, rz=176.058, shoulder=lefty, elbow=epositive, wrist=wpositive, fatherId=fReference[0]}
  [5726] = {x=528.674, y=-248.986, z=66, rx=-180, rz=175.86, shoulder=lefty, elbow=epositive, wrist=wpositive, fatherId=fReference[0]}
  [5727] = {x=530.086, y=-248.884, z=66, rx=180, rz=175.662, shoulder=lefty, elbow=epositive, wrist=wpositive, fatherId=fReference[0]}
  [5728] = {x=531.498, y=-248.777, z=66, rx=-180, rz=175.465, shoulder=lefty, elbow=epositive, wrist=wpositive, fatherId=fReference[0]}
  [5729] = {x=532.911, y=-248.665, z=66, rx=-180, rz=175.267, shoulder=lefty, elbow=epositive, wrist=wpositive, fatherId=fReference[0]}
  [5730] = {x=534.323, y=-248.548, z=66, rx=-180, rz=175.07, shoulder=lefty, elbow=epositive, wrist=wpositive, fatherId=fReference[0]}
  [5731] = {x=535.734, y=-248.426, z=66, rx=-180, rz=174.874, shoulder=lefty, elbow=epositive, wrist=wpositive, fatherId=fReference[0]}
  [5732] = {x=537.146, y=-248.3, z=66, rx=-180, rz=174.677, shoulder=lefty, elbow=epositive, wrist=wpositive, fatherId=fReference[0]}
  [5733] = {x=538.557, y=-248.168, z=66, rx=-180, rz=174.481, shoulder=lefty, elbow=epositive, wrist=wpositive, fatherId=fReference[0]}
  [5734] = {x=539.968, y=-248.032, z=66, rx=180, rz=174.285, shoulder=lefty, elbow=epositive, wrist=wpositive, fatherId=fReference[0]}
  [5735] = {x=541.379, y=-247.891, z=66, rx=-180, rz=174.089, shoulder=lefty, elbow=epositive, wrist=wpositive, fatherId=fReference[0]}
  [5736] = {x=542.79, y=-247.744, z=66, rx=-180, rz=173.894, shoulder=lefty, elbow=epositive, wrist=wpositive, fatherId=fReference[0]}
  [5737] = {x=544.2, y=-247.594, z=66, rx=-180, rz=173.698, shoulder=lefty, elbow=epositive, wrist=wpositive, fatherId=fReference[0]}
  [5738] = {x=545.61, y=-247.438, z=66, rx=-180, rz=173.504, shoulder=lefty, elbow=epositive, wrist=wpositive, fatherId=fReference[0]}
  [5739] = {x=547.02, y=-247.277, z=66, rx=180, rz=173.309, shoulder=lefty, elbow=epositive, wrist=wpositive, fatherId=fReference[0]}
  [5740] = {x=548.43, y=-247.112, z=66, rx=-180, rz=173.115, shoulder=lefty, elbow=epositive, wrist=wpositive, fatherId=fReference[0]}
  [5741] = {x=549.839, y=-246.942, z=66, rx=180, rz=172.921, shoulder=lefty, elbow=epositive, wrist=wpositive, fatherId=fReference[0]}
  [5742] = {x=551.248, y=-246.767, z=66, rx=-180, rz=172.727, shoulder=lefty, elbow=epositive, wrist=wpositive, fatherId=fReference[0]}
  [5743] = {x=552.657, y=-246.587, z=66, rx=-180, rz=172.534, shoulder=lefty, elbow=epositive, wrist=wpositive, fatherId=fReference[0]}
  [5744] = {x=554.065, y=-246.402, z=66, rx=-180, rz=172.341, shoulder=lefty, elbow=epositive, wrist=wpositive, fatherId=fReference[0]}
  [5745] = {x=555.473, y=-246.213, z=66, rx=180, rz=172.149, shoulder=lefty, elbow=epositive, wrist=wpositive, fatherId=fReference[0]}
  [5746] = {x=556.881, y=-246.019, z=66, rx=-180, rz=171.957, shoulder=lefty, elbow=epositive, wrist=wpositive, fatherId=fReference[0]}
  [5747] = {x=558.289, y=-245.82, z=66, rx=180, rz=171.765, shoulder=lefty, elbow=epositive, wrist=wpositive, fatherId=fReference[0]}
  [5748] = {x=559.696, y=-245.616, z=66, rx=-180, rz=171.574, shoulder=lefty, elbow=epositive, wrist=wpositive, fatherId=fReference[0]}
  [5749] = {x=561.102, y=-245.408, z=66, rx=-180, rz=171.383, shoulder=lefty, elbow=epositive, wrist=wpositive, fatherId=fReference[0]}
  [5750] = {x=562.509, y=-245.195, z=66, rx=-180, rz=171.192, shoulder=lefty, elbow=epositive, wrist=wpositive, fatherId=fReference[0]}
  [5751] = {x=563.915, y=-244.977, z=66, rx=180, rz=171.002, shoulder=lefty, elbow=epositive, wrist=wpositive, fatherId=fReference[0]}
  [5752] = {x=565.321, y=-244.755, z=66, rx=-180, rz=170.813, shoulder=lefty, elbow=epositive, wrist=wpositive, fatherId=fReference[0]}
  [5753] = {x=566.726, y=-244.527, z=66, rx=-180, rz=170.623, shoulder=lefty, elbow=epositive, wrist=wpositive, fatherId=fReference[0]}
  [5754] = {x=568.131, y=-244.295, z=66, rx=180, rz=170.435, shoulder=lefty, elbow=epositive, wrist=wpositive, fatherId=fReference[0]}
  [5755] = {x=569.535, y=-244.059, z=66, rx=180, rz=170.246, shoulder=lefty, elbow=epositive, wrist=wpositive, fatherId=fReference[0]}
  [5756] = {x=570.939, y=-243.817, z=66, rx=-180, rz=170.058, shoulder=lefty, elbow=epositive, wrist=wpositive, fatherId=fReference[0]}
  [5757] = {x=572.343, y=-243.571, z=66, rx=-180, rz=169.871, shoulder=lefty, elbow=epositive, wrist=wpositive, fatherId=fReference[0]}
  [5758] = {x=573.746, y=-243.32, z=66, rx=-180, rz=169.684, shoulder=lefty, elbow=epositive, wrist=wpositive, fatherId=fReference[0]}
  [5759] = {x=575.149, y=-243.065, z=66, rx=180, rz=169.497, shoulder=lefty, elbow=epositive, wrist=wpositive, fatherId=fReference[0]}
  [5760] = {x=576.552, y=-242.805, z=66, rx=-180, rz=169.311, shoulder=lefty, elbow=epositive, wrist=wpositive, fatherId=fReference[0]}
  [5761] = {x=577.954, y=-242.54, z=66, rx=-180, rz=169.126, shoulder=lefty, elbow=epositive, wrist=wpositive, fatherId=fReference[0]}
  [5762] = {x=579.355, y=-242.271, z=66, rx=180, rz=168.941, shoulder=lefty, elbow=epositive, wrist=wpositive, fatherId=fReference[0]}
  [5763] = {x=580.757, y=-241.997, z=66, rx=-180, rz=168.756, shoulder=lefty, elbow=epositive, wrist=wpositive, fatherId=fReference[0]}
  [5764] = {x=582.157, y=-241.719, z=66, rx=-180, rz=168.572, shoulder=lefty, elbow=epositive, wrist=wpositive, fatherId=fReference[0]}
  [5765] = {x=583.557, y=-241.436, z=66, rx=-180, rz=168.389, shoulder=lefty, elbow=epositive, wrist=wpositive, fatherId=fReference[0]}
  [5766] = {x=584.957, y=-241.148, z=66, rx=180, rz=168.206, shoulder=lefty, elbow=epositive, wrist=wpositive, fatherId=fReference[0]}
  [5767] = {x=586.357, y=-240.856, z=66, rx=180, rz=168.023, shoulder=lefty, elbow=epositive, wrist=wpositive, fatherId=fReference[0]}
  [5768] = {x=587.755, y=-240.559, z=66, rx=180, rz=167.841, shoulder=lefty, elbow=epositive, wrist=wpositive, fatherId=fReference[0]}
  [5769] = {x=589.154, y=-240.258, z=66, rx=-180, rz=167.66, shoulder=lefty, elbow=epositive, wrist=wpositive, fatherId=fReference[0]}
  [5770] = {x=590.552, y=-239.952, z=66, rx=180, rz=167.479, shoulder=lefty, elbow=epositive, wrist=wpositive, fatherId=fReference[0]}
  [5771] = {x=591.949, y=-239.642, z=66, rx=180, rz=167.299, shoulder=lefty, elbow=epositive, wrist=wpositive, fatherId=fReference[0]}
  [5772] = {x=593.346, y=-239.327, z=66, rx=180, rz=167.119, shoulder=lefty, elbow=epositive, wrist=wpositive, fatherId=fReference[0]}
  [5773] = {x=594.742, y=-239.008, z=66, rx=180, rz=166.94, shoulder=lefty, elbow=epositive, wrist=wpositive, fatherId=fReference[0]}
  [5774] = {x=596.138, y=-238.684, z=66, rx=-180, rz=166.761, shoulder=lefty, elbow=epositive, wrist=wpositive, fatherId=fReference[0]}
  [5775] = {x=597.533, y=-238.356, z=66, rx=180, rz=166.583, shoulder=lefty, elbow=epositive, wrist=wpositive, fatherId=fReference[0]}
  [5776] = {x=598.928, y=-238.023, z=66, rx=180, rz=166.405, shoulder=lefty, elbow=epositive, wrist=wpositive, fatherId=fReference[0]}
  [5777] = {x=600.322, y=-237.686, z=66, rx=-180, rz=166.229, shoulder=lefty, elbow=epositive, wrist=wpositive, fatherId=fReference[0]}
  [5778] = {x=601.716, y=-237.344, z=66, rx=-180, rz=166.052, shoulder=lefty, elbow=epositive, wrist=wpositive, fatherId=fReference[0]}
  [5779] = {x=603.109, y=-236.998, z=66, rx=180, rz=165.877, shoulder=lefty, elbow=epositive, wrist=wpositive, fatherId=fReference[0]}
  [5780] = {x=604.502, y=-236.648, z=66, rx=-180, rz=165.702, shoulder=lefty, elbow=epositive, wrist=wpositive, fatherId=fReference[0]}
  [5781] = {x=605.894, y=-236.293, z=66, rx=-180, rz=165.527, shoulder=lefty, elbow=epositive, wrist=wpositive, fatherId=fReference[0]}
  [5782] = {x=607.286, y=-235.934, z=66, rx=-180, rz=165.353, shoulder=lefty, elbow=epositive, wrist=wpositive, fatherId=fReference[0]}
  [5783] = {x=608.677, y=-235.57, z=66, rx=-180, rz=165.18, shoulder=lefty, elbow=epositive, wrist=wpositive, fatherId=fReference[0]}
  [5784] = {x=610.067, y=-235.202, z=66, rx=-180, rz=165.007, shoulder=lefty, elbow=epositive, wrist=wpositive, fatherId=fReference[0]}
  [5785] = {x=611.457, y=-234.83, z=66, rx=180, rz=164.835, shoulder=lefty, elbow=epositive, wrist=wpositive, fatherId=fReference[0]}
  [5786] = {x=612.846, y=-234.454, z=66, rx=-180, rz=164.664, shoulder=lefty, elbow=epositive, wrist=wpositive, fatherId=fReference[0]}
  [5787] = {x=614.235, y=-234.073, z=66, rx=-180, rz=164.493, shoulder=lefty, elbow=epositive, wrist=wpositive, fatherId=fReference[0]}
  [5788] = {x=615.623, y=-233.688, z=66, rx=-180, rz=164.323, shoulder=lefty, elbow=epositive, wrist=wpositive, fatherId=fReference[0]}
  [5789] = {x=617.01, y=-233.298, z=66, rx=180, rz=164.153, shoulder=lefty, elbow=epositive, wrist=wpositive, fatherId=fReference[0]}
  [5790] = {x=618.397, y=-232.905, z=66, rx=180, rz=163.985, shoulder=lefty, elbow=epositive, wrist=wpositive, fatherId=fReference[0]}
  [5791] = {x=619.783, y=-232.507, z=66, rx=-180, rz=163.816, shoulder=lefty, elbow=epositive, wrist=wpositive, fatherId=fReference[0]}
  [5792] = {x=621.169, y=-232.104, z=66, rx=180, rz=163.649, shoulder=lefty, elbow=epositive, wrist=wpositive, fatherId=fReference[0]}
  [5793] = {x=622.554, y=-231.698, z=66, rx=180, rz=163.482, shoulder=lefty, elbow=epositive, wrist=wpositive, fatherId=fReference[0]}
  [5794] = {x=623.939, y=-231.288, z=66, rx=-180, rz=163.316, shoulder=lefty, elbow=epositive, wrist=wpositive, fatherId=fReference[0]}
  [5795] = {x=625.322, y=-230.873, z=66, rx=180, rz=163.15, shoulder=lefty, elbow=epositive, wrist=wpositive, fatherId=fReference[0]}
  [5796] = {x=626.706, y=-230.454, z=66, rx=-180, rz=162.985, shoulder=lefty, elbow=epositive, wrist=wpositive, fatherId=fReference[0]}
  [5797] = {x=628.088, y=-230.031, z=66, rx=-180, rz=162.821, shoulder=lefty, elbow=epositive, wrist=wpositive, fatherId=fReference[0]}
  [5798] = {x=629.47, y=-229.604, z=66, rx=-180, rz=162.657, shoulder=lefty, elbow=epositive, wrist=wpositive, fatherId=fReference[0]}
  [5799] = {x=630.851, y=-229.172, z=66, rx=-180, rz=162.494, shoulder=lefty, elbow=epositive, wrist=wpositive, fatherId=fReference[0]}
  [5800] = {x=632.232, y=-228.737, z=66, rx=-180, rz=162.332, shoulder=lefty, elbow=epositive, wrist=wpositive, fatherId=fReference[0]}
  [5801] = {x=633.612, y=-228.297, z=66, rx=-180, rz=162.171, shoulder=lefty, elbow=epositive, wrist=wpositive, fatherId=fReference[0]}
  [5802] = {x=634.991, y=-227.854, z=66, rx=-180, rz=162.01, shoulder=lefty, elbow=epositive, wrist=wpositive, fatherId=fReference[0]}
  [5803] = {x=636.37, y=-227.406, z=66, rx=180, rz=161.85, shoulder=lefty, elbow=epositive, wrist=wpositive, fatherId=fReference[0]}
  [5804] = {x=637.748, y=-226.954, z=66, rx=-180, rz=161.69, shoulder=lefty, elbow=epositive, wrist=wpositive, fatherId=fReference[0]}
  [5805] = {x=639.125, y=-226.498, z=66, rx=180, rz=161.531, shoulder=lefty, elbow=epositive, wrist=wpositive, fatherId=fReference[0]}
  [5806] = {x=640.502, y=-226.038, z=66, rx=180, rz=161.373, shoulder=lefty, elbow=epositive, wrist=wpositive, fatherId=fReference[0]}
  [5807] = {x=641.878, y=-225.575, z=66, rx=180, rz=161.216, shoulder=lefty, elbow=epositive, wrist=wpositive, fatherId=fReference[0]}
  [5808] = {x=643.254, y=-225.107, z=66, rx=180, rz=161.059, shoulder=lefty, elbow=epositive, wrist=wpositive, fatherId=fReference[0]}
  [5809] = {x=644.628, y=-224.635, z=66, rx=180, rz=160.903, shoulder=lefty, elbow=epositive, wrist=wpositive, fatherId=fReference[0]}
  [5810] = {x=646.002, y=-224.159, z=66, rx=180, rz=160.748, shoulder=lefty, elbow=epositive, wrist=wpositive, fatherId=fReference[0]}
  [5811] = {x=647.376, y=-223.68, z=66, rx=-180, rz=160.593, shoulder=lefty, elbow=epositive, wrist=wpositive, fatherId=fReference[0]}
  [5812] = {x=648.748, y=-223.196, z=66, rx=-180, rz=160.439, shoulder=lefty, elbow=epositive, wrist=wpositive, fatherId=fReference[0]}
  [5813] = {x=650.12, y=-222.709, z=66, rx=-180, rz=160.286, shoulder=lefty, elbow=epositive, wrist=wpositive, fatherId=fReference[0]}
  [5814] = {x=651.491, y=-222.217, z=66, rx=180, rz=160.133, shoulder=lefty, elbow=epositive, wrist=wpositive, fatherId=fReference[0]}
  [5815] = {x=652.862, y=-221.722, z=66, rx=-180, rz=159.981, shoulder=lefty, elbow=epositive, wrist=wpositive, fatherId=fReference[0]}
  [5816] = {x=654.232, y=-221.223, z=66, rx=-180, rz=159.83, shoulder=lefty, elbow=epositive, wrist=wpositive, fatherId=fReference[0]}
  [5817] = {x=655.601, y=-220.72, z=66, rx=180, rz=159.68, shoulder=lefty, elbow=epositive, wrist=wpositive, fatherId=fReference[0]}
  [5818] = {x=656.969, y=-220.213, z=66, rx=-180, rz=159.53, shoulder=lefty, elbow=epositive, wrist=wpositive, fatherId=fReference[0]}
  [5819] = {x=658.337, y=-219.703, z=66, rx=180, rz=159.381, shoulder=lefty, elbow=epositive, wrist=wpositive, fatherId=fReference[0]}
  [5820] = {x=659.704, y=-219.189, z=66, rx=-180, rz=159.233, shoulder=lefty, elbow=epositive, wrist=wpositive, fatherId=fReference[0]}
  [5821] = {x=661.07, y=-218.67, z=66, rx=180, rz=159.086, shoulder=lefty, elbow=epositive, wrist=wpositive, fatherId=fReference[0]}
  [5822] = {x=662.436, y=-218.149, z=66, rx=180, rz=158.939, shoulder=lefty, elbow=epositive, wrist=wpositive, fatherId=fReference[0]}
  [5823] = {x=663.801, y=-217.623, z=66, rx=180, rz=158.793, shoulder=lefty, elbow=epositive, wrist=wpositive, fatherId=fReference[0]}
  [5824] = {x=665.165, y=-217.094, z=66, rx=180, rz=158.647, shoulder=lefty, elbow=epositive, wrist=wpositive, fatherId=fReference[0]}
  [5825] = {x=666.528, y=-216.561, z=66, rx=180, rz=158.503, shoulder=lefty, elbow=epositive, wrist=wpositive, fatherId=fReference[0]}
  [5826] = {x=667.891, y=-216.024, z=66, rx=180, rz=158.359, shoulder=lefty, elbow=epositive, wrist=wpositive, fatherId=fReference[0]}
  [5827] = {x=669.253, y=-215.484, z=66, rx=180, rz=158.216, shoulder=lefty, elbow=epositive, wrist=wpositive, fatherId=fReference[0]}
  [5828] = {x=670.614, y=-214.94, z=66, rx=180, rz=158.073, shoulder=lefty, elbow=epositive, wrist=wpositive, fatherId=fReference[0]}
  [5829] = {x=671.974, y=-214.392, z=66, rx=180, rz=157.931, shoulder=lefty, elbow=epositive, wrist=wpositive, fatherId=fReference[0]}
  [5830] = {x=673.334, y=-213.841, z=66, rx=-180, rz=157.79, shoulder=lefty, elbow=epositive, wrist=wpositive, fatherId=fReference[0]}
  [5831] = {x=674.693, y=-213.286, z=66, rx=-180, rz=157.65, shoulder=lefty, elbow=epositive, wrist=wpositive, fatherId=fReference[0]}
  [5832] = {x=676.052, y=-212.727, z=66, rx=180, rz=157.51, shoulder=lefty, elbow=epositive, wrist=wpositive, fatherId=fReference[0]}
  [5833] = {x=677.409, y=-212.165, z=66, rx=180, rz=157.371, shoulder=lefty, elbow=epositive, wrist=wpositive, fatherId=fReference[0]}
  [5834] = {x=678.766, y=-211.6, z=66, rx=180, rz=157.233, shoulder=lefty, elbow=epositive, wrist=wpositive, fatherId=fReference[0]}
  [5835] = {x=680.122, y=-211.031, z=66, rx=180, rz=157.096, shoulder=lefty, elbow=epositive, wrist=wpositive, fatherId=fReference[0]}
  [5836] = {x=681.477, y=-210.458, z=66, rx=-180, rz=156.959, shoulder=lefty, elbow=epositive, wrist=wpositive, fatherId=fReference[0]}
  [5837] = {x=682.832, y=-209.882, z=66, rx=180, rz=156.823, shoulder=lefty, elbow=epositive, wrist=wpositive, fatherId=fReference[0]}
  [5838] = {x=684.186, y=-209.302, z=66, rx=180, rz=156.688, shoulder=lefty, elbow=epositive, wrist=wpositive, fatherId=fReference[0]}
  [5839] = {x=685.539, y=-208.719, z=66, rx=-180, rz=156.553, shoulder=lefty, elbow=epositive, wrist=wpositive, fatherId=fReference[0]}
  [5840] = {x=686.891, y=-208.133, z=66, rx=-180, rz=156.42, shoulder=lefty, elbow=epositive, wrist=wpositive, fatherId=fReference[0]}
  [5841] = {x=688.243, y=-207.543, z=66, rx=180, rz=156.287, shoulder=lefty, elbow=epositive, wrist=wpositive, fatherId=fReference[0]}
  [5842] = {x=689.593, y=-206.949, z=66, rx=-180, rz=156.154, shoulder=lefty, elbow=epositive, wrist=wpositive, fatherId=fReference[0]}
  [5843] = {x=690.943, y=-206.353, z=66, rx=180, rz=156.023, shoulder=lefty, elbow=epositive, wrist=wpositive, fatherId=fReference[0]}
  [5844] = {x=692.293, y=-205.753, z=66, rx=-180, rz=155.892, shoulder=lefty, elbow=epositive, wrist=wpositive, fatherId=fReference[0]}
  [5845] = {x=693.641, y=-205.149, z=66, rx=-180, rz=155.762, shoulder=lefty, elbow=epositive, wrist=wpositive, fatherId=fReference[0]}
  [5846] = {x=694.989, y=-204.542, z=66, rx=180, rz=155.632, shoulder=lefty, elbow=epositive, wrist=wpositive, fatherId=fReference[0]}
  [5847] = {x=696.336, y=-203.932, z=66, rx=180, rz=155.503, shoulder=lefty, elbow=epositive, wrist=wpositive, fatherId=fReference[0]}
  [5848] = {x=697.682, y=-203.319, z=66, rx=-180, rz=155.375, shoulder=lefty, elbow=epositive, wrist=wpositive, fatherId=fReference[0]}
  [5849] = {x=699.028, y=-202.702, z=66, rx=-180, rz=155.248, shoulder=lefty, elbow=epositive, wrist=wpositive, fatherId=fReference[0]}
  [5850] = {x=700.373, y=-202.082, z=66, rx=180, rz=155.122, shoulder=lefty, elbow=epositive, wrist=wpositive, fatherId=fReference[0]}
  [5851] = {x=701.717, y=-201.459, z=66, rx=180, rz=154.996, shoulder=lefty, elbow=epositive, wrist=wpositive, fatherId=fReference[0]}
  [5852] = {x=703.06, y=-200.832, z=66, rx=-180, rz=154.871, shoulder=lefty, elbow=epositive, wrist=wpositive, fatherId=fReference[0]}
  [5853] = {x=704.403, y=-200.203, z=66, rx=-180, rz=154.746, shoulder=lefty, elbow=epositive, wrist=wpositive, fatherId=fReference[0]}
  [5854] = {x=705.744, y=-199.57, z=66, rx=180, rz=154.622, shoulder=lefty, elbow=epositive, wrist=wpositive, fatherId=fReference[0]}
  [5855] = {x=707.085, y=-198.933, z=66, rx=180, rz=154.499, shoulder=lefty, elbow=epositive, wrist=wpositive, fatherId=fReference[0]}
  [5856] = {x=708.426, y=-198.294, z=66, rx=180, rz=154.377, shoulder=lefty, elbow=epositive, wrist=wpositive, fatherId=fReference[0]}
  [5857] = {x=709.765, y=-197.652, z=66, rx=-180, rz=154.256, shoulder=lefty, elbow=epositive, wrist=wpositive, fatherId=fReference[0]}
  [5858] = {x=711.104, y=-197.006, z=66, rx=180, rz=154.135, shoulder=lefty, elbow=epositive, wrist=wpositive, fatherId=fReference[0]}
  [5859] = {x=712.442, y=-196.357, z=66, rx=-180, rz=154.015, shoulder=lefty, elbow=epositive, wrist=wpositive, fatherId=fReference[0]}
  [5860] = {x=713.779, y=-195.706, z=66, rx=180, rz=153.895, shoulder=lefty, elbow=epositive, wrist=wpositive, fatherId=fReference[0]}
  [5861] = {x=715.116, y=-195.051, z=66, rx=180, rz=153.776, shoulder=lefty, elbow=epositive, wrist=wpositive, fatherId=fReference[0]}
  [5862] = {x=716.452, y=-194.393, z=66, rx=180, rz=153.658, shoulder=lefty, elbow=epositive, wrist=wpositive, fatherId=fReference[0]}
  [5863] = {x=717.787, y=-193.732, z=66, rx=180, rz=153.541, shoulder=lefty, elbow=epositive, wrist=wpositive, fatherId=fReference[0]}
  [5864] = {x=719.121, y=-193.067, z=66, rx=180, rz=153.424, shoulder=lefty, elbow=epositive, wrist=wpositive, fatherId=fReference[0]}
  [5865] = {x=720.455, y=-192.4, z=66, rx=-180, rz=153.309, shoulder=lefty, elbow=epositive, wrist=wpositive, fatherId=fReference[0]}
  [5866] = {x=721.788, y=-191.73, z=66, rx=-180, rz=153.193, shoulder=lefty, elbow=epositive, wrist=wpositive, fatherId=fReference[0]}
  [5867] = {x=723.12, y=-191.057, z=66, rx=-180, rz=153.079, shoulder=lefty, elbow=epositive, wrist=wpositive, fatherId=fReference[0]}
  [5868] = {x=724.451, y=-190.381, z=66, rx=-180, rz=152.965, shoulder=lefty, elbow=epositive, wrist=wpositive, fatherId=fReference[0]}
  [5869] = {x=725.782, y=-189.702, z=66, rx=-180, rz=152.852, shoulder=lefty, elbow=epositive, wrist=wpositive, fatherId=fReference[0]}
  [5870] = {x=727.112, y=-189.02, z=66, rx=180, rz=152.739, shoulder=lefty, elbow=epositive, wrist=wpositive, fatherId=fReference[0]}
  [5871] = {x=728.441, y=-188.335, z=66, rx=-180, rz=152.628, shoulder=lefty, elbow=epositive, wrist=wpositive, fatherId=fReference[0]}
  [5872] = {x=729.77, y=-187.647, z=66, rx=180, rz=152.517, shoulder=lefty, elbow=epositive, wrist=wpositive, fatherId=fReference[0]}
  [5873] = {x=731.098, y=-186.957, z=66, rx=-180, rz=152.406, shoulder=lefty, elbow=epositive, wrist=wpositive, fatherId=fReference[0]}
  [5874] = {x=732.425, y=-186.263, z=66, rx=180, rz=152.297, shoulder=lefty, elbow=epositive, wrist=wpositive, fatherId=fReference[0]}
  [5875] = {x=733.751, y=-185.567, z=66, rx=-180, rz=152.188, shoulder=lefty, elbow=epositive, wrist=wpositive, fatherId=fReference[0]}
  [5876] = {x=735.077, y=-184.867, z=66, rx=180, rz=152.079, shoulder=lefty, elbow=epositive, wrist=wpositive, fatherId=fReference[0]}
  [5877] = {x=736.401, y=-184.165, z=66, rx=-180, rz=151.972, shoulder=lefty, elbow=epositive, wrist=wpositive, fatherId=fReference[0]}
  [5878] = {x=737.726, y=-183.46, z=66, rx=180, rz=151.865, shoulder=lefty, elbow=epositive, wrist=wpositive, fatherId=fReference[0]}
  [5879] = {x=739.049, y=-182.753, z=66, rx=180, rz=151.759, shoulder=lefty, elbow=epositive, wrist=wpositive, fatherId=fReference[0]}
  [5880] = {x=740.372, y=-182.042, z=66, rx=-180, rz=151.653, shoulder=lefty, elbow=epositive, wrist=wpositive, fatherId=fReference[0]}
  [5881] = {x=741.694, y=-181.329, z=66, rx=180, rz=151.548, shoulder=lefty, elbow=epositive, wrist=wpositive, fatherId=fReference[0]}
  [5882] = {x=743.015, y=-180.613, z=66, rx=-180, rz=151.444, shoulder=lefty, elbow=epositive, wrist=wpositive, fatherId=fReference[0]}
  [5883] = {x=744.336, y=-179.894, z=66, rx=180, rz=151.341, shoulder=lefty, elbow=epositive, wrist=wpositive, fatherId=fReference[0]}
  [5884] = {x=745.656, y=-179.173, z=66, rx=180, rz=151.238, shoulder=lefty, elbow=epositive, wrist=wpositive, fatherId=fReference[0]}
  [5885] = {x=746.975, y=-178.449, z=66, rx=180, rz=151.136, shoulder=lefty, elbow=epositive, wrist=wpositive, fatherId=fReference[0]}
  [5886] = {x=748.293, y=-177.722, z=66, rx=180, rz=151.034, shoulder=lefty, elbow=epositive, wrist=wpositive, fatherId=fReference[0]}
  [5887] = {x=749.611, y=-176.993, z=66, rx=180, rz=150.933, shoulder=lefty, elbow=epositive, wrist=wpositive, fatherId=fReference[0]}
  [5888] = {x=750.928, y=-176.26, z=66, rx=-180, rz=150.833, shoulder=lefty, elbow=epositive, wrist=wpositive, fatherId=fReference[0]}
  [5889] = {x=752.244, y=-175.526, z=66, rx=180, rz=150.734, shoulder=lefty, elbow=epositive, wrist=wpositive, fatherId=fReference[0]}
  [5890] = {x=753.56, y=-174.788, z=66, rx=180, rz=150.635, shoulder=lefty, elbow=epositive, wrist=wpositive, fatherId=fReference[0]}
  [5891] = {x=754.875, y=-174.049, z=66, rx=180, rz=150.537, shoulder=lefty, elbow=epositive, wrist=wpositive, fatherId=fReference[0]}
  [5892] = {x=756.189, y=-173.306, z=66, rx=-180, rz=150.439, shoulder=lefty, elbow=epositive, wrist=wpositive, fatherId=fReference[0]}
  [5893] = {x=757.503, y=-172.561, z=66, rx=180, rz=150.342, shoulder=lefty, elbow=epositive, wrist=wpositive, fatherId=fReference[0]}
  [5894] = {x=758.816, y=-171.814, z=66, rx=180, rz=150.246, shoulder=lefty, elbow=epositive, wrist=wpositive, fatherId=fReference[0]}
  [5895] = {x=760.128, y=-171.064, z=66, rx=180, rz=150.151, shoulder=lefty, elbow=epositive, wrist=wpositive, fatherId=fReference[0]}
  [5896] = {x=761.439, y=-170.311, z=66, rx=180, rz=150.056, shoulder=lefty, elbow=epositive, wrist=wpositive, fatherId=fReference[0]}
  [5897] = {x=762.75, y=-169.556, z=66, rx=180, rz=149.961, shoulder=lefty, elbow=epositive, wrist=wpositive, fatherId=fReference[0]}
  [5898] = {x=764.06, y=-168.798, z=66, rx=180, rz=149.868, shoulder=lefty, elbow=epositive, wrist=wpositive, fatherId=fReference[0]}
  [5899] = {x=765.369, y=-168.038, z=66, rx=180, rz=149.775, shoulder=lefty, elbow=epositive, wrist=wpositive, fatherId=fReference[0]}
  [5900] = {x=766.678, y=-167.276, z=66, rx=180, rz=149.683, shoulder=lefty, elbow=epositive, wrist=wpositive, fatherId=fReference[0]}
  [5901] = {x=767.986, y=-166.511, z=66, rx=-180, rz=149.591, shoulder=lefty, elbow=epositive, wrist=wpositive, fatherId=fReference[0]}
  [5902] = {x=769.293, y=-165.744, z=66, rx=180, rz=149.5, shoulder=lefty, elbow=epositive, wrist=wpositive, fatherId=fReference[0]}
  [5903] = {x=770.6, y=-164.974, z=66, rx=180, rz=149.41, shoulder=lefty, elbow=epositive, wrist=wpositive, fatherId=fReference[0]}
  [5904] = {x=771.906, y=-164.202, z=66, rx=180, rz=149.32, shoulder=lefty, elbow=epositive, wrist=wpositive, fatherId=fReference[0]}
  [5905] = {x=773.211, y=-163.428, z=66, rx=180, rz=149.231, shoulder=lefty, elbow=epositive, wrist=wpositive, fatherId=fReference[0]}
  [5906] = {x=774.516, y=-162.651, z=66, rx=-180, rz=149.142, shoulder=lefty, elbow=epositive, wrist=wpositive, fatherId=fReference[0]}
  [5907] = {x=775.82, y=-161.872, z=66, rx=-180, rz=149.054, shoulder=lefty, elbow=epositive, wrist=wpositive, fatherId=fReference[0]}
  [5908] = {x=777.123, y=-161.091, z=66, rx=-180, rz=148.967, shoulder=lefty, elbow=epositive, wrist=wpositive, fatherId=fReference[0]}
  [5909] = {x=778.425, y=-160.307, z=66, rx=180, rz=148.881, shoulder=lefty, elbow=epositive, wrist=wpositive, fatherId=fReference[0]}
  [5910] = {x=779.727, y=-159.521, z=66, rx=180, rz=148.795, shoulder=lefty, elbow=epositive, wrist=wpositive, fatherId=fReference[0]}
  [5911] = {x=781.028, y=-158.733, z=66, rx=-180, rz=148.709, shoulder=lefty, elbow=epositive, wrist=wpositive, fatherId=fReference[0]}
  [5912] = {x=782.329, y=-157.942, z=66, rx=180, rz=148.625, shoulder=lefty, elbow=epositive, wrist=wpositive, fatherId=fReference[0]}
  [5913] = {x=783.629, y=-157.15, z=66, rx=180, rz=148.54, shoulder=lefty, elbow=epositive, wrist=wpositive, fatherId=fReference[0]}
  [5914] = {x=784.928, y=-156.355, z=66, rx=-180, rz=148.457, shoulder=lefty, elbow=epositive, wrist=wpositive, fatherId=fReference[0]}
  [5915] = {x=786.227, y=-155.558, z=66, rx=180, rz=148.374, shoulder=lefty, elbow=epositive, wrist=wpositive, fatherId=fReference[0]}
  [5916] = {x=787.524, y=-154.758, z=66, rx=180, rz=148.292, shoulder=lefty, elbow=epositive, wrist=wpositive, fatherId=fReference[0]}
  [5917] = {x=788.822, y=-153.957, z=66, rx=180, rz=148.21, shoulder=lefty, elbow=epositive, wrist=wpositive, fatherId=fReference[0]}
  [5918] = {x=790.118, y=-153.153, z=66, rx=180, rz=148.129, shoulder=lefty, elbow=epositive, wrist=wpositive, fatherId=fReference[0]}
  [5919] = {x=791.414, y=-152.348, z=66, rx=180, rz=148.049, shoulder=lefty, elbow=epositive, wrist=wpositive, fatherId=fReference[0]}
  [5920] = {x=792.709, y=-151.54, z=66, rx=-180, rz=147.969, shoulder=lefty, elbow=epositive, wrist=wpositive, fatherId=fReference[0]}
  [5921] = {x=794.004, y=-150.73, z=66, rx=180, rz=147.89, shoulder=lefty, elbow=epositive, wrist=wpositive, fatherId=fReference[0]}
  [5922] = {x=795.298, y=-149.918, z=66, rx=180, rz=147.811, shoulder=lefty, elbow=epositive, wrist=wpositive, fatherId=fReference[0]}
  [5923] = {x=796.591, y=-149.104, z=66, rx=180, rz=147.733, shoulder=lefty, elbow=epositive, wrist=wpositive, fatherId=fReference[0]}
  [5924] = {x=797.884, y=-148.288, z=66, rx=-180, rz=147.656, shoulder=lefty, elbow=epositive, wrist=wpositive, fatherId=fReference[0]}
  [5925] = {x=799.175, y=-147.47, z=66, rx=180, rz=147.579, shoulder=lefty, elbow=epositive, wrist=wpositive, fatherId=fReference[0]}
  [5926] = {x=800.467, y=-146.65, z=66, rx=180, rz=147.503, shoulder=lefty, elbow=epositive, wrist=wpositive, fatherId=fReference[0]}
  [5927] = {x=801.757, y=-145.827, z=66, rx=180, rz=147.427, shoulder=lefty, elbow=epositive, wrist=wpositive, fatherId=fReference[0]}
  [5928] = {x=803.047, y=-145.003, z=66, rx=-180, rz=147.352, shoulder=lefty, elbow=epositive, wrist=wpositive, fatherId=fReference[0]}
  [5929] = {x=804.337, y=-144.177, z=66, rx=-180, rz=147.277, shoulder=lefty, elbow=epositive, wrist=wpositive, fatherId=fReference[0]}
  [5930] = {x=805.626, y=-143.349, z=66, rx=180, rz=147.204, shoulder=lefty, elbow=epositive, wrist=wpositive, fatherId=fReference[0]}
  [5931] = {x=806.914, y=-142.519, z=66, rx=180, rz=147.13, shoulder=lefty, elbow=epositive, wrist=wpositive, fatherId=fReference[0]}
  [5932] = {x=808.201, y=-141.687, z=66, rx=-180, rz=147.058, shoulder=lefty, elbow=epositive, wrist=wpositive, fatherId=fReference[0]}
  [5933] = {x=809.488, y=-140.853, z=66, rx=-180, rz=146.986, shoulder=lefty, elbow=epositive, wrist=wpositive, fatherId=fReference[0]}
  [5934] = {x=810.774, y=-140.017, z=66, rx=180, rz=146.914, shoulder=lefty, elbow=epositive, wrist=wpositive, fatherId=fReference[0]}
  [5935] = {x=812.06, y=-139.18, z=66, rx=180, rz=146.843, shoulder=lefty, elbow=epositive, wrist=wpositive, fatherId=fReference[0]}
  [5936] = {x=813.345, y=-138.34, z=66, rx=-180, rz=146.773, shoulder=lefty, elbow=epositive, wrist=wpositive, fatherId=fReference[0]}
  [5937] = {x=814.629, y=-137.499, z=66, rx=180, rz=146.703, shoulder=lefty, elbow=epositive, wrist=wpositive, fatherId=fReference[0]}
  [5938] = {x=815.913, y=-136.656, z=66, rx=-180, rz=146.634, shoulder=lefty, elbow=epositive, wrist=wpositive, fatherId=fReference[0]}
  [5939] = {x=817.196, y=-135.811, z=66, rx=-180, rz=146.565, shoulder=lefty, elbow=epositive, wrist=wpositive, fatherId=fReference[0]}
  [5940] = {x=818.479, y=-134.964, z=66, rx=-180, rz=146.497, shoulder=lefty, elbow=epositive, wrist=wpositive, fatherId=fReference[0]}
  [5941] = {x=819.761, y=-134.115, z=66, rx=180, rz=146.429, shoulder=lefty, elbow=epositive, wrist=wpositive, fatherId=fReference[0]}
  [5942] = {x=821.042, y=-133.265, z=66, rx=180, rz=146.362, shoulder=lefty, elbow=epositive, wrist=wpositive, fatherId=fReference[0]}
  [5943] = {x=822.323, y=-132.413, z=66, rx=-180, rz=146.296, shoulder=lefty, elbow=epositive, wrist=wpositive, fatherId=fReference[0]}
  [5944] = {x=823.603, y=-131.559, z=66, rx=180, rz=146.23, shoulder=lefty, elbow=epositive, wrist=wpositive, fatherId=fReference[0]}
  [5945] = {x=824.882, y=-130.703, z=66, rx=180, rz=146.165, shoulder=lefty, elbow=epositive, wrist=wpositive, fatherId=fReference[0]}
  [5946] = {x=826.161, y=-129.846, z=66, rx=180, rz=146.1, shoulder=lefty, elbow=epositive, wrist=wpositive, fatherId=fReference[0]}
  [5947] = {x=827.44, y=-128.987, z=66, rx=-180, rz=146.036, shoulder=lefty, elbow=epositive, wrist=wpositive, fatherId=fReference[0]}
  [5948] = {x=828.717, y=-128.127, z=66, rx=-180, rz=145.972, shoulder=lefty, elbow=epositive, wrist=wpositive, fatherId=fReference[0]}
  [5949] = {x=829.994, y=-127.264, z=66, rx=180, rz=145.909, shoulder=lefty, elbow=epositive, wrist=wpositive, fatherId=fReference[0]}
  [5950] = {x=831.271, y=-126.4, z=66, rx=-180, rz=145.847, shoulder=lefty, elbow=epositive, wrist=wpositive, fatherId=fReference[0]}
  [5951] = {x=832.547, y=-125.535, z=66, rx=180, rz=145.785, shoulder=lefty, elbow=epositive, wrist=wpositive, fatherId=fReference[0]}
  [5952] = {x=833.822, y=-124.667, z=66, rx=180, rz=145.723, shoulder=lefty, elbow=epositive, wrist=wpositive, fatherId=fReference[0]}
  [5953] = {x=835.097, y=-123.798, z=66, rx=-180, rz=145.662, shoulder=lefty, elbow=epositive, wrist=wpositive, fatherId=fReference[0]}
  [5954] = {x=836.372, y=-122.928, z=66, rx=180, rz=145.602, shoulder=lefty, elbow=epositive, wrist=wpositive, fatherId=fReference[0]}
  [5955] = {x=837.645, y=-122.056, z=66, rx=180, rz=145.542, shoulder=lefty, elbow=epositive, wrist=wpositive, fatherId=fReference[0]}
  [5956] = {x=838.918, y=-121.182, z=66, rx=180, rz=145.483, shoulder=lefty, elbow=epositive, wrist=wpositive, fatherId=fReference[0]}
  [5957] = {x=840.191, y=-120.307, z=66, rx=-180, rz=145.424, shoulder=lefty, elbow=epositive, wrist=wpositive, fatherId=fReference[0]}
  [5958] = {x=841.463, y=-119.43, z=66, rx=-180, rz=145.366, shoulder=lefty, elbow=epositive, wrist=wpositive, fatherId=fReference[0]}
  [5959] = {x=842.734, y=-118.552, z=66, rx=180, rz=145.308, shoulder=lefty, elbow=epositive, wrist=wpositive, fatherId=fReference[0]}
  [5960] = {x=844.005, y=-117.672, z=66, rx=180, rz=145.251, shoulder=lefty, elbow=epositive, wrist=wpositive, fatherId=fReference[0]}
  [5961] = {x=845.276, y=-116.791, z=66, rx=-180, rz=145.195, shoulder=lefty, elbow=epositive, wrist=wpositive, fatherId=fReference[0]}
  [5962] = {x=846.545, y=-115.908, z=66, rx=180, rz=145.139, shoulder=lefty, elbow=epositive, wrist=wpositive, fatherId=fReference[0]}
  [5963] = {x=847.815, y=-115.024, z=66, rx=180, rz=145.083, shoulder=lefty, elbow=epositive, wrist=wpositive, fatherId=fReference[0]}
  [5964] = {x=849.084, y=-114.139, z=66, rx=-180, rz=145.028, shoulder=lefty, elbow=epositive, wrist=wpositive, fatherId=fReference[0]}
  [5965] = {x=850.352, y=-113.251, z=66, rx=-180, rz=144.974, shoulder=lefty, elbow=epositive, wrist=wpositive, fatherId=fReference[0]}
  [5966] = {x=851.619, y=-112.363, z=66, rx=-180, rz=144.92, shoulder=lefty, elbow=epositive, wrist=wpositive, fatherId=fReference[0]}
  [5967] = {x=852.887, y=-111.473, z=66, rx=180, rz=144.866, shoulder=lefty, elbow=epositive, wrist=wpositive, fatherId=fReference[0]}
  [5968] = {x=854.153, y=-110.582, z=66, rx=-180, rz=144.813, shoulder=lefty, elbow=epositive, wrist=wpositive, fatherId=fReference[0]}
  [5969] = {x=855.419, y=-109.689, z=66, rx=180, rz=144.761, shoulder=lefty, elbow=epositive, wrist=wpositive, fatherId=fReference[0]}
  [5970] = {x=856.685, y=-108.795, z=66, rx=-180, rz=144.709, shoulder=lefty, elbow=epositive, wrist=wpositive, fatherId=fReference[0]}
  [5971] = {x=857.95, y=-107.899, z=66, rx=180, rz=144.657, shoulder=lefty, elbow=epositive, wrist=wpositive, fatherId=fReference[0]}
  [5972] = {x=859.215, y=-107.003, z=66, rx=180, rz=144.607, shoulder=lefty, elbow=epositive, wrist=wpositive, fatherId=fReference[0]}
  [5973] = {x=860.479, y=-106.104, z=66, rx=-180, rz=144.556, shoulder=lefty, elbow=epositive, wrist=wpositive, fatherId=fReference[0]}
  [5974] = {x=861.742, y=-105.205, z=66, rx=180, rz=144.506, shoulder=lefty, elbow=epositive, wrist=wpositive, fatherId=fReference[0]}
  [5975] = {x=863.006, y=-104.304, z=66, rx=180, rz=144.457, shoulder=lefty, elbow=epositive, wrist=wpositive, fatherId=fReference[0]}
  [5976] = {x=864.268, y=-103.402, z=66, rx=-180, rz=144.408, shoulder=lefty, elbow=epositive, wrist=wpositive, fatherId=fReference[0]}
  [5977] = {x=865.53, y=-102.499, z=66, rx=-180, rz=144.36, shoulder=lefty, elbow=epositive, wrist=wpositive, fatherId=fReference[0]}
  [5978] = {x=866.792, y=-101.594, z=66, rx=180, rz=144.312, shoulder=lefty, elbow=epositive, wrist=wpositive, fatherId=fReference[0]}
  [5979] = {x=868.053, y=-100.688, z=66, rx=180, rz=144.265, shoulder=lefty, elbow=epositive, wrist=wpositive, fatherId=fReference[0]}
